LREAL#19.579149162561258, LREAL#19.593929605703352, LREAL#19.608190954002232, LREAL#19.62195143826828, LREAL#19.635228649038805, LREAL#19.648039559064692, LREAL#19.660400545007292, LREAL#19.672327408373313, LREAL#19.683835395714475, LREAL#19.694939218117742, LREAL#19.705653070011053, LREAL#19.715990647308583, LREAL#19.725965164918737, LREAL#19.735589373637257, LREAL#19.74487557644704, LREAL#19.753835644245491, LREAL#19.762481031019547, LREAL#19.77082278848771, LREAL#19.778871580227889, LREAL#19.786637695309036, LREAL#19.794131061444048, LREAL#18.854802175821771, LREAL#18.895021963501684, LREAL#18.933829216781984, LREAL#18.971273544413613, LREAL#19.00740281286912, LREAL#19.042263207532141, LREAL#19.075899291737894, LREAL#19.108354063740133, LREAL#19.13966901167742, LREAL#19.169884166608945, LREAL#19.199038153687717, LREAL#19.227168241536525, LREAL#19.25431038988981, LREAL#19.280499295562311, LREAL#19.305768436803309, LREAL#19.330150116093094, LREAL#19.353675501436445, LREAL#19.37637466620583, LREAL#19.398276627585318, LREAL#19.419409383664327, LREAL#19.439799949228611, LREAL#19.459474390294268, LREAL#19.478457857428893, LREAL#19.496774617902481, LREAL#19.514448086709184, LREAL#19.531500856499555, LREAL#19.54795472646158, LREAL#19.563830730187384, LREAL#19.579149162561258, LREAL#19.593929605703352, LREAL#19.608190954002232, LREAL#19.62195143826828, LREAL#19.635228649038805, LREAL#19.648039559064692, LREAL#19.660400545007292, LREAL#19.672327408373313, LREAL#19.683835395714475, LREAL#19.694939218117742, LREAL#19.705653070011053, LREAL#19.715990647308583, LREAL#19.725965164918737, LREAL#19.735589373637257, LREAL#19.74487557644704, LREAL#19.753835644245491, LREAL#19.762481031019547, LREAL#19.77082278848771, LREAL#19.778871580227889, LREAL#19.786637695309036, LREAL#19.794131061444048, LREAL#19.801361257680728, LREAL#18.895021963501684, LREAL#18.933829216781984, LREAL#18.971273544413613, LREAL#19.00740281286912, LREAL#19.042263207532141, LREAL#19.075899291737894, LREAL#19.108354063740133, LREAL#19.13966901167742, LREAL#19.169884166608945, LREAL#19.199038153687717, LREAL#19.227168241536525, LREAL#19.25431038988981, LREAL#19.280499295562311, LREAL#19.305768436803309, LREAL#19.330150116093094, LREAL#19.353675501436445, LREAL#19.37637466620583, LREAL#19.398276627585318, LREAL#19.419409383664327, LREAL#19.439799949228611, LREAL#19.459474390294268, LREAL#19.478457857428893, LREAL#19.496774617902481, LREAL#19.514448086709184, LREAL#19.531500856499555, LREAL#19.54795472646158, LREAL#19.563830730187384, LREAL#19.579149162561258, LREAL#19.593929605703352, LREAL#19.608190954002232, LREAL#19.62195143826828, LREAL#19.635228649038805, LREAL#19.648039559064692, LREAL#19.660400545007292, LREAL#19.672327408373313, LREAL#19.683835395714475, LREAL#19.694939218117742, LREAL#19.705653070011053, LREAL#19.715990647308583, LREAL#19.725965164918737, LREAL#19.735589373637257, LREAL#19.74487557644704, LREAL#19.753835644245491, LREAL#19.762481031019547, LREAL#19.77082278848771, LREAL#19.778871580227889, LREAL#19.786637695309036, LREAL#19.794131061444048, LREAL#19.801361257680728, LREAL#19.808337526647041, LREAL#18.933829216781984, LREAL#18.971273544413613, LREAL#19.00740281286912, LREAL#19.042263207532141, LREAL#19.075899291737894, LREAL#19.108354063740133, LREAL#19.13966901167742, LREAL#19.169884166608945, LREAL#19.199038153687717, LREAL#19.227168241536525, LREAL#19.25431038988981, LREAL#19.280499295562311, LREAL#19.305768436803309, LREAL#19.330150116093094, LREAL#19.353675501436445, LREAL#19.37637466620583, LREAL#19.398276627585318, LREAL#19.419409383664327, LREAL#19.439799949228611, LREAL#19.459474390294268, LREAL#19.478457857428893, LREAL#19.496774617902481, LREAL#19.514448086709184, LREAL#19.531500856499555, LREAL#19.54795472646158, LREAL#19.563830730187384, LREAL#19.579149162561258, LREAL#19.593929605703352, LREAL#19.608190954002232, LREAL#19.62195143826828, LREAL#19.635228649038805, LREAL#19.648039559064692, LREAL#19.660400545007292, LREAL#19.672327408373313, LREAL#19.683835395714475, LREAL#19.694939218117742, LREAL#19.705653070011053, LREAL#19.715990647308583, LREAL#19.725965164918737, LREAL#19.735589373637257, LREAL#19.74487557644704, LREAL#19.753835644245491, LREAL#19.762481031019547, LREAL#19.77082278848771, LREAL#19.778871580227889, LREAL#19.786637695309036, LREAL#19.794131061444048, LREAL#19.801361257680728, LREAL#19.808337526647041, LREAL#19.815068786366307, LREAL#18.971273544413613, LREAL#19.00740281286912, LREAL#19.042263207532141, LREAL#19.075899291737894, LREAL#19.108354063740133, LREAL#19.13966901167742, LREAL#19.169884166608945, LREAL#19.199038153687717, LREAL#19.227168241536525, LREAL#19.25431038988981, LREAL#19.280499295562311, LREAL#19.305768436803309, LREAL#19.330150116093094, LREAL#19.353675501436445, LREAL#19.37637466620583, LREAL#19.398276627585318, LREAL#19.419409383664327, LREAL#19.439799949228611, LREAL#19.459474390294268, LREAL#19.478457857428893, LREAL#19.496774617902481, LREAL#19.514448086709184, LREAL#19.531500856499555, LREAL#19.54795472646158, LREAL#19.563830730187384, LREAL#19.579149162561258, LREAL#19.593929605703352, LREAL#19.608190954002232, LREAL#19.62195143826828, LREAL#19.635228649038805, LREAL#19.648039559064692, LREAL#19.660400545007292, LREAL#19.672327408373313, LREAL#19.683835395714475, LREAL#19.694939218117742, LREAL#19.705653070011053, LREAL#19.715990647308583, LREAL#19.725965164918737, LREAL#19.735589373637257, LREAL#19.74487557644704, LREAL#19.753835644245491, LREAL#19.762481031019547, LREAL#19.77082278848771, LREAL#19.778871580227889, LREAL#19.786637695309036, LREAL#19.794131061444048, LREAL#19.801361257680728, LREAL#19.808337526647041, LREAL#19.815068786366307, LREAL#19.821563641657438, LREAL#19.00740281286912, LREAL#19.042263207532141, LREAL#19.075899291737894, LREAL#19.108354063740133, LREAL#19.13966901167742, LREAL#19.169884166608945, LREAL#19.199038153687717, LREAL#19.227168241536525, LREAL#19.25431038988981, LREAL#19.280499295562311, LREAL#19.305768436803309, LREAL#19.330150116093094, LREAL#19.353675501436445, LREAL#19.37637466620583, LREAL#19.398276627585318, LREAL#19.419409383664327, LREAL#19.439799949228611, LREAL#19.459474390294268, LREAL#19.478457857428893, LREAL#19.496774617902481, LREAL#19.514448086709184, LREAL#19.531500856499555, LREAL#19.54795472646158, LREAL#19.563830730187384, LREAL#19.579149162561258, LREAL#19.593929605703352, LREAL#19.608190954002232, LREAL#19.62195143826828, LREAL#19.635228649038805, LREAL#19.648039559064692, LREAL#19.660400545007292, LREAL#19.672327408373313, LREAL#19.683835395714475, LREAL#19.694939218117742, LREAL#19.705653070011053, LREAL#19.715990647308583, LREAL#19.725965164918737, LREAL#19.735589373637257, LREAL#19.74487557644704, LREAL#19.753835644245491, LREAL#19.762481031019547, LREAL#19.77082278848771, LREAL#19.778871580227889, LREAL#19.786637695309036, LREAL#19.794131061444048, LREAL#19.801361257680728, LREAL#19.808337526647041, LREAL#19.815068786366307, LREAL#19.821563641657438, LREAL#19.827830395134797, LREAL#19.042263207532141, LREAL#19.075899291737894, LREAL#19.108354063740133, LREAL#19.13966901167742, LREAL#19.169884166608945, LREAL#19.199038153687717, LREAL#19.227168241536525, LREAL#19.25431038988981, LREAL#19.280499295562311, LREAL#19.305768436803309, LREAL#19.330150116093094, LREAL#19.353675501436445, LREAL#19.37637466620583, LREAL#19.398276627585318, LREAL#19.419409383664327, LREAL#19.439799949228611, LREAL#19.459474390294268, LREAL#19.478457857428893, LREAL#19.496774617902481, LREAL#19.514448086709184, LREAL#19.531500856499555, LREAL#19.54795472646158, LREAL#19.563830730187384, LREAL#19.579149162561258, LREAL#19.593929605703352, LREAL#19.608190954002232, LREAL#19.62195143826828, LREAL#19.635228649038805, LREAL#19.648039559064692, LREAL#19.660400545007292, LREAL#19.672327408373313, LREAL#19.683835395714475, LREAL#19.694939218117742, LREAL#19.705653070011053, LREAL#19.715990647308583, LREAL#19.725965164918737, LREAL#19.735589373637257, LREAL#19.74487557644704, LREAL#19.753835644245491, LREAL#19.762481031019547, LREAL#19.77082278848771, LREAL#19.778871580227889, LREAL#19.786637695309036, LREAL#19.794131061444048, LREAL#19.801361257680728, LREAL#19.808337526647041, LREAL#19.815068786366307, LREAL#19.821563641657438, LREAL#19.827830395134797, LREAL#19.833877057821745, LREAL#19.075899291737894, LREAL#19.108354063740133, LREAL#19.13966901167742, LREAL#19.169884166608945, LREAL#19.199038153687717, LREAL#19.227168241536525, LREAL#19.25431038988981, LREAL#19.280499295562311, LREAL#19.305768436803309, LREAL#19.330150116093094, LREAL#19.353675501436445, LREAL#19.37637466620583, LREAL#19.398276627585318, LREAL#19.419409383664327, LREAL#19.439799949228611, LREAL#19.459474390294268, LREAL#19.478457857428893, LREAL#19.496774617902481, LREAL#19.514448086709184, LREAL#19.531500856499555, LREAL#19.54795472646158, LREAL#19.563830730187384, LREAL#19.579149162561258, LREAL#19.593929605703352, LREAL#19.608190954002232, LREAL#19.62195143826828, LREAL#19.635228649038805, LREAL#19.648039559064692, LREAL#19.660400545007292, LREAL#19.672327408373313, LREAL#19.683835395714475, LREAL#19.694939218117742, LREAL#19.705653070011053, LREAL#19.715990647308583, LREAL#19.725965164918737, LREAL#19.735589373637257, LREAL#19.74487557644704, LREAL#19.753835644245491, LREAL#19.762481031019547, LREAL#19.77082278848771, LREAL#19.778871580227889, LREAL#19.786637695309036, LREAL#19.794131061444048, LREAL#19.801361257680728, LREAL#19.808337526647041, LREAL#19.815068786366307, LREAL#19.821563641657438, LREAL#19.827830395134797, LREAL#19.833877057821745, LREAL#19.839711359391419, LREAL#19.108354063740133, LREAL#19.13966901167742, LREAL#19.169884166608945, LREAL#19.199038153687717, LREAL#19.227168241536525, LREAL#19.25431038988981, LREAL#19.280499295562311, LREAL#19.305768436803309, LREAL#19.330150116093094, LREAL#19.353675501436445, LREAL#19.37637466620583, LREAL#19.398276627585318, LREAL#19.419409383664327, LREAL#19.439799949228611, LREAL#19.459474390294268, LREAL#19.478457857428893, LREAL#19.496774617902481, LREAL#19.514448086709184, LREAL#19.531500856499555, LREAL#19.54795472646158, LREAL#19.563830730187384, LREAL#19.579149162561258, LREAL#19.593929605703352, LREAL#19.608190954002232, LREAL#19.62195143826828, LREAL#19.635228649038805, LREAL#19.648039559064692, LREAL#19.660400545007292, LREAL#19.672327408373313, LREAL#19.683835395714475, LREAL#19.694939218117742, LREAL#19.705653070011053, LREAL#19.715990647308583, LREAL#19.725965164918737, LREAL#19.735589373637257, LREAL#19.74487557644704, LREAL#19.753835644245491, LREAL#19.762481031019547, LREAL#19.77082278848771, LREAL#19.778871580227889, LREAL#19.786637695309036, LREAL#19.794131061444048, LREAL#19.801361257680728, LREAL#19.808337526647041, LREAL#19.815068786366307, LREAL#19.821563641657438, LREAL#19.827830395134797, LREAL#19.833877057821745, LREAL#19.839711359391419, LREAL#19.845340758047868, LREAL#19.13966901167742, LREAL#19.169884166608945, LREAL#19.199038153687717, LREAL#19.227168241536525, LREAL#19.25431038988981, LREAL#19.280499295562311, LREAL#19.305768436803309, LREAL#19.330150116093094, LREAL#19.353675501436445, LREAL#19.37637466620583, LREAL#19.398276627585318, LREAL#19.419409383664327, LREAL#19.439799949228611, LREAL#19.459474390294268, LREAL#19.478457857428893, LREAL#19.496774617902481, LREAL#19.514448086709184, LREAL#19.531500856499555, LREAL#19.54795472646158, LREAL#19.563830730187384, LREAL#19.579149162561258, LREAL#19.593929605703352, LREAL#19.608190954002232, LREAL#19.62195143826828, LREAL#19.635228649038805, LREAL#19.648039559064692, LREAL#19.660400545007292, LREAL#19.672327408373313, LREAL#19.683835395714475, LREAL#19.694939218117742, LREAL#19.705653070011053, LREAL#19.715990647308583, LREAL#19.725965164918737, LREAL#19.735589373637257, LREAL#19.74487557644704, LREAL#19.753835644245491, LREAL#19.762481031019547, LREAL#19.77082278848771, LREAL#19.778871580227889, LREAL#19.786637695309036, LREAL#19.794131061444048, LREAL#19.801361257680728, LREAL#19.808337526647041, LREAL#19.815068786366307, LREAL#19.821563641657438, LREAL#19.827830395134797, LREAL#19.833877057821745, LREAL#19.839711359391419, LREAL#19.845340758047868, LREAL#19.850772450060148, LREAL#19.169884166608945, LREAL#19.199038153687717, LREAL#19.227168241536525, LREAL#19.25431038988981, LREAL#19.280499295562311, LREAL#19.305768436803309, LREAL#19.330150116093094, LREAL#19.353675501436445, LREAL#19.37637466620583, LREAL#19.398276627585318, LREAL#19.419409383664327, LREAL#19.439799949228611, LREAL#19.459474390294268, LREAL#19.478457857428893, LREAL#19.496774617902481, LREAL#19.514448086709184, LREAL#19.531500856499555, LREAL#19.54795472646158, LREAL#19.563830730187384, LREAL#19.579149162561258, LREAL#19.593929605703352, LREAL#19.608190954002232, LREAL#19.62195143826828, LREAL#19.635228649038805, LREAL#19.648039559064692, LREAL#19.660400545007292, LREAL#19.672327408373313, LREAL#19.683835395714475, LREAL#19.694939218117742, LREAL#19.705653070011053, LREAL#19.715990647308583, LREAL#19.725965164918737, LREAL#19.735589373637257, LREAL#19.74487557644704, LREAL#19.753835644245491, LREAL#19.762481031019547, LREAL#19.77082278848771, LREAL#19.778871580227889, LREAL#19.786637695309036, LREAL#19.794131061444048, LREAL#19.801361257680728, LREAL#19.808337526647041, LREAL#19.815068786366307, LREAL#19.821563641657438, LREAL#19.827830395134797, LREAL#19.833877057821745, LREAL#19.839711359391419, LREAL#19.845340758047868, LREAL#19.850772450060148, LREAL#19.856013378961581, LREAL#19.199038153687717, LREAL#19.227168241536525, LREAL#19.25431038988981, LREAL#19.280499295562311, LREAL#19.305768436803309, LREAL#19.330150116093094, LREAL#19.353675501436445, LREAL#19.37637466620583, LREAL#19.398276627585318, LREAL#19.419409383664327, LREAL#19.439799949228611, LREAL#19.459474390294268, LREAL#19.478457857428893, LREAL#19.496774617902481, LREAL#19.514448086709184, LREAL#19.531500856499555, LREAL#19.54795472646158, LREAL#19.563830730187384, LREAL#19.579149162561258, LREAL#19.593929605703352, LREAL#19.608190954002232, LREAL#19.62195143826828, LREAL#19.635228649038805, LREAL#19.648039559064692, LREAL#19.660400545007292, LREAL#19.672327408373313, LREAL#19.683835395714475, LREAL#19.694939218117742, LREAL#19.705653070011053, LREAL#19.715990647308583, LREAL#19.725965164918737, LREAL#19.735589373637257, LREAL#19.74487557644704, LREAL#19.753835644245491, LREAL#19.762481031019547, LREAL#19.77082278848771, LREAL#19.778871580227889, LREAL#19.786637695309036, LREAL#19.794131061444048, LREAL#19.801361257680728, LREAL#19.808337526647041, LREAL#19.815068786366307, LREAL#19.821563641657438, LREAL#19.827830395134797, LREAL#19.833877057821745, LREAL#19.839711359391419, LREAL#19.845340758047868, LREAL#19.850772450060148, LREAL#19.856013378961581, LREAL#19.861070244425928, LREAL#19.227168241536525, LREAL#19.25431038988981, LREAL#19.280499295562311, LREAL#19.305768436803309, LREAL#19.330150116093094, LREAL#19.353675501436445, LREAL#19.37637466620583, LREAL#19.398276627585318, LREAL#19.419409383664327, LREAL#19.439799949228611, LREAL#19.459474390294268, LREAL#19.478457857428893, LREAL#19.496774617902481, LREAL#19.514448086709184, LREAL#19.531500856499555, LREAL#19.54795472646158, LREAL#19.563830730187384, LREAL#19.579149162561258, LREAL#19.593929605703352, LREAL#19.608190954002232, LREAL#19.62195143826828, LREAL#19.635228649038805, LREAL#19.648039559064692, LREAL#19.660400545007292, LREAL#19.672327408373313, LREAL#19.683835395714475, LREAL#19.694939218117742, LREAL#19.705653070011053, LREAL#19.715990647308583, LREAL#19.725965164918737, LREAL#19.735589373637257, LREAL#19.74487557644704, LREAL#19.753835644245491, LREAL#19.762481031019547, LREAL#19.77082278848771, LREAL#19.778871580227889, LREAL#19.786637695309036, LREAL#19.794131061444048, LREAL#19.801361257680728, LREAL#19.808337526647041, LREAL#19.815068786366307, LREAL#19.821563641657438, LREAL#19.827830395134797, LREAL#19.833877057821745, LREAL#19.839711359391419, LREAL#19.845340758047868, LREAL#19.850772450060148, LREAL#19.856013378961581, LREAL#19.861070244425928, LREAL#19.865949510831836, LREAL#19.25431038988981, LREAL#19.280499295562311, LREAL#19.305768436803309, LREAL#19.330150116093094, LREAL#19.353675501436445, LREAL#19.37637466620583, LREAL#19.398276627585318, LREAL#19.419409383664327, LREAL#19.439799949228611, LREAL#19.459474390294268, LREAL#19.478457857428893, LREAL#19.496774617902481, LREAL#19.514448086709184, LREAL#19.531500856499555, LREAL#19.54795472646158, LREAL#19.563830730187384, LREAL#19.579149162561258, LREAL#19.593929605703352, LREAL#19.608190954002232, LREAL#19.62195143826828, LREAL#19.635228649038805, LREAL#19.648039559064692, LREAL#19.660400545007292, LREAL#19.672327408373313, LREAL#19.683835395714475, LREAL#19.694939218117742, LREAL#19.705653070011053, LREAL#19.715990647308583, LREAL#19.725965164918737, LREAL#19.735589373637257, LREAL#19.74487557644704, LREAL#19.753835644245491, LREAL#19.762481031019547, LREAL#19.77082278848771, LREAL#19.778871580227889, LREAL#19.786637695309036, LREAL#19.794131061444048, LREAL#19.801361257680728, LREAL#19.808337526647041, LREAL#19.815068786366307, LREAL#19.821563641657438, LREAL#19.827830395134797, LREAL#19.833877057821745, LREAL#19.839711359391419, LREAL#19.845340758047868, LREAL#19.850772450060148, LREAL#19.856013378961581, LREAL#19.861070244425928, LREAL#19.865949510831836, LREAL#19.870657415526487, LREAL#19.280499295562311, LREAL#19.305768436803309, LREAL#19.330150116093094, LREAL#19.353675501436445, LREAL#19.37637466620583, LREAL#19.398276627585318, LREAL#19.419409383664327, LREAL#19.439799949228611, LREAL#19.459474390294268, LREAL#19.478457857428893, LREAL#19.496774617902481, LREAL#19.514448086709184, LREAL#19.531500856499555, LREAL#19.54795472646158, LREAL#19.563830730187384, LREAL#19.579149162561258, LREAL#19.593929605703352, LREAL#19.608190954002232, LREAL#19.62195143826828, LREAL#19.635228649038805, LREAL#19.648039559064692, LREAL#19.660400545007292, LREAL#19.672327408373313, LREAL#19.683835395714475, LREAL#19.694939218117742, LREAL#19.705653070011053, LREAL#19.715990647308583, LREAL#19.725965164918737, LREAL#19.735589373637257, LREAL#19.74487557644704, LREAL#19.753835644245491, LREAL#19.762481031019547, LREAL#19.77082278848771, LREAL#19.778871580227889, LREAL#19.786637695309036, LREAL#19.794131061444048, LREAL#19.801361257680728, LREAL#19.808337526647041, LREAL#19.815068786366307, LREAL#19.821563641657438, LREAL#19.827830395134797, LREAL#19.833877057821745, LREAL#19.839711359391419, LREAL#19.845340758047868, LREAL#19.850772450060148, LREAL#19.856013378961581, LREAL#19.861070244425928, LREAL#19.865949510831836, LREAL#19.870657415526487, LREAL#19.875199976799031, LREAL#19.305768436803309, LREAL#19.330150116093094, LREAL#19.353675501436445, LREAL#19.37637466620583, LREAL#19.398276627585318, LREAL#19.419409383664327, LREAL#19.439799949228611, LREAL#19.459474390294268, LREAL#19.478457857428893, LREAL#19.496774617902481, LREAL#19.514448086709184, LREAL#19.531500856499555, LREAL#19.54795472646158, LREAL#19.563830730187384, LREAL#19.579149162561258, LREAL#19.593929605703352, LREAL#19.608190954002232, LREAL#19.62195143826828, LREAL#19.635228649038805, LREAL#19.648039559064692, LREAL#19.660400545007292, LREAL#19.672327408373313, LREAL#19.683835395714475, LREAL#19.694939218117742, LREAL#19.705653070011053, LREAL#19.715990647308583, LREAL#19.725965164918737, LREAL#19.735589373637257, LREAL#19.74487557644704, LREAL#19.753835644245491, LREAL#19.762481031019547, LREAL#19.77082278848771, LREAL#19.778871580227889, LREAL#19.786637695309036, LREAL#19.794131061444048, LREAL#19.801361257680728, LREAL#19.808337526647041, LREAL#19.815068786366307, LREAL#19.821563641657438, LREAL#19.827830395134797, LREAL#19.833877057821745, LREAL#19.839711359391419, LREAL#19.845340758047868, LREAL#19.850772450060148, LREAL#19.856013378961581, LREAL#19.861070244425928, LREAL#19.865949510831836, LREAL#19.870657415526487, LREAL#19.875199976799031, LREAL#19.879583001573998, LREAL#19.330150116093094, LREAL#19.353675501436445, LREAL#19.37637466620583, LREAL#19.398276627585318, LREAL#19.419409383664327, LREAL#19.439799949228611, LREAL#19.459474390294268, LREAL#19.478457857428893, LREAL#19.496774617902481, LREAL#19.514448086709184, LREAL#19.531500856499555, LREAL#19.54795472646158, LREAL#19.563830730187384, LREAL#19.579149162561258, LREAL#19.593929605703352, LREAL#19.608190954002232, LREAL#19.62195143826828, LREAL#19.635228649038805, LREAL#19.648039559064692, LREAL#19.660400545007292, LREAL#19.672327408373313, LREAL#19.683835395714475, LREAL#19.694939218117742, LREAL#19.705653070011053, LREAL#19.715990647308583, LREAL#19.725965164918737, LREAL#19.735589373637257, LREAL#19.74487557644704, LREAL#19.753835644245491, LREAL#19.762481031019547, LREAL#19.77082278848771, LREAL#19.778871580227889, LREAL#19.786637695309036, LREAL#19.794131061444048, LREAL#19.801361257680728, LREAL#19.808337526647041, LREAL#19.815068786366307, LREAL#19.821563641657438, LREAL#19.827830395134797, LREAL#19.833877057821745, LREAL#19.839711359391419, LREAL#19.845340758047868, LREAL#19.850772450060148, LREAL#19.856013378961581, LREAL#19.861070244425928, LREAL#19.865949510831836, LREAL#19.870657415526487, LREAL#19.875199976799031, LREAL#19.879583001573998, LREAL#19.883812092834489, LREAL#19.353675501436445, LREAL#19.37637466620583, LREAL#19.398276627585318, LREAL#19.419409383664327, LREAL#19.439799949228611, LREAL#19.459474390294268, LREAL#19.478457857428893, LREAL#19.496774617902481, LREAL#19.514448086709184, LREAL#19.531500856499555, LREAL#19.54795472646158, LREAL#19.563830730187384, LREAL#19.579149162561258, LREAL#19.593929605703352, LREAL#19.608190954002232, LREAL#19.62195143826828, LREAL#19.635228649038805, LREAL#19.648039559064692, LREAL#19.660400545007292, LREAL#19.672327408373313, LREAL#19.683835395714475, LREAL#19.694939218117742, LREAL#19.705653070011053, LREAL#19.715990647308583, LREAL#19.725965164918737, LREAL#19.735589373637257, LREAL#19.74487557644704, LREAL#19.753835644245491, LREAL#19.762481031019547, LREAL#19.77082278848771, LREAL#19.778871580227889, LREAL#19.786637695309036, LREAL#19.794131061444048, LREAL#19.801361257680728, LREAL#19.808337526647041, LREAL#19.815068786366307, LREAL#19.821563641657438, LREAL#19.827830395134797, LREAL#19.833877057821745, LREAL#19.839711359391419, LREAL#19.845340758047868, LREAL#19.850772450060148, LREAL#19.856013378961581, LREAL#19.861070244425928, LREAL#19.865949510831836, LREAL#19.870657415526487, LREAL#19.875199976799031, LREAL#19.879583001573998, LREAL#19.883812092834489, LREAL#19.88789265678469, LREAL#19.37637466620583, LREAL#19.398276627585318, LREAL#19.419409383664327, LREAL#19.439799949228611, LREAL#19.459474390294268, LREAL#19.478457857428893, LREAL#19.496774617902481, LREAL#19.514448086709184, LREAL#19.531500856499555, LREAL#19.54795472646158, LREAL#19.563830730187384, LREAL#19.579149162561258, LREAL#19.593929605703352, LREAL#19.608190954002232, LREAL#19.62195143826828, LREAL#19.635228649038805, LREAL#19.648039559064692, LREAL#19.660400545007292, LREAL#19.672327408373313, LREAL#19.683835395714475, LREAL#19.694939218117742, LREAL#19.705653070011053, LREAL#19.715990647308583, LREAL#19.725965164918737, LREAL#19.735589373637257, LREAL#19.74487557644704, LREAL#19.753835644245491, LREAL#19.762481031019547, LREAL#19.77082278848771, LREAL#19.778871580227889, LREAL#19.786637695309036, LREAL#19.794131061444048, LREAL#19.801361257680728, LREAL#19.808337526647041, LREAL#19.815068786366307, LREAL#19.821563641657438, LREAL#19.827830395134797, LREAL#19.833877057821745, LREAL#19.839711359391419, LREAL#19.845340758047868, LREAL#19.850772450060148, LREAL#19.856013378961581, LREAL#19.861070244425928, LREAL#19.865949510831836, LREAL#19.870657415526487, LREAL#19.875199976799031, LREAL#19.879583001573998, LREAL#19.883812092834489, LREAL#19.88789265678469, LREAL#19.891829909760816, LREAL#19.398276627585318, LREAL#19.419409383664327, LREAL#19.439799949228611, LREAL#19.459474390294268, LREAL#19.478457857428893, LREAL#19.496774617902481, LREAL#19.514448086709184, LREAL#19.531500856499555, LREAL#19.54795472646158, LREAL#19.563830730187384, LREAL#19.579149162561258, LREAL#19.593929605703352, LREAL#19.608190954002232, LREAL#19.62195143826828, LREAL#19.635228649038805, LREAL#19.648039559064692, LREAL#19.660400545007292, LREAL#19.672327408373313, LREAL#19.683835395714475, LREAL#19.694939218117742, LREAL#19.705653070011053, LREAL#19.715990647308583, LREAL#19.725965164918737, LREAL#19.735589373637257, LREAL#19.74487557644704, LREAL#19.753835644245491, LREAL#19.762481031019547, LREAL#19.77082278848771, LREAL#19.778871580227889, LREAL#19.786637695309036, LREAL#19.794131061444048, LREAL#19.801361257680728, LREAL#19.808337526647041, LREAL#19.815068786366307, LREAL#19.821563641657438, LREAL#19.827830395134797, LREAL#19.833877057821745, LREAL#19.839711359391419, LREAL#19.845340758047868, LREAL#19.850772450060148, LREAL#19.856013378961581, LREAL#19.861070244425928, LREAL#19.865949510831836, LREAL#19.870657415526487, LREAL#19.875199976799031, LREAL#19.879583001573998, LREAL#19.883812092834489, LREAL#19.88789265678469, LREAL#19.891829909760816, LREAL#19.895628884899349, LREAL#19.419409383664327, LREAL#19.439799949228611, LREAL#19.459474390294268, LREAL#19.478457857428893, LREAL#19.496774617902481, LREAL#19.514448086709184, LREAL#19.531500856499555, LREAL#19.54795472646158, LREAL#19.563830730187384, LREAL#19.579149162561258, LREAL#19.593929605703352, LREAL#19.608190954002232, LREAL#19.62195143826828, LREAL#19.635228649038805, LREAL#19.648039559064692, LREAL#19.660400545007292, LREAL#19.672327408373313, LREAL#19.683835395714475, LREAL#19.694939218117742, LREAL#19.705653070011053, LREAL#19.715990647308583, LREAL#19.725965164918737, LREAL#19.735589373637257, LREAL#19.74487557644704, LREAL#19.753835644245491, LREAL#19.762481031019547, LREAL#19.77082278848771, LREAL#19.778871580227889, LREAL#19.786637695309036, LREAL#19.794131061444048, LREAL#19.801361257680728, LREAL#19.808337526647041, LREAL#19.815068786366307, LREAL#19.821563641657438, LREAL#19.827830395134797, LREAL#19.833877057821745, LREAL#19.839711359391419, LREAL#19.845340758047868, LREAL#19.850772450060148, LREAL#19.856013378961581, LREAL#19.861070244425928, LREAL#19.865949510831836, LREAL#19.870657415526487, LREAL#19.875199976799031, LREAL#19.879583001573998, LREAL#19.883812092834489, LREAL#19.88789265678469, LREAL#19.891829909760816, LREAL#19.895628884899349, LREAL#19.899294438571086, LREAL#19.439799949228611, LREAL#19.459474390294268, LREAL#19.478457857428893, LREAL#19.496774617902481, LREAL#19.514448086709184, LREAL#19.531500856499555, LREAL#19.54795472646158, LREAL#19.563830730187384, LREAL#19.579149162561258, LREAL#19.593929605703352, LREAL#19.608190954002232, LREAL#19.62195143826828, LREAL#19.635228649038805, LREAL#19.648039559064692, LREAL#19.660400545007292, LREAL#19.672327408373313, LREAL#19.683835395714475, LREAL#19.694939218117742, LREAL#19.705653070011053, LREAL#19.715990647308583, LREAL#19.725965164918737, LREAL#19.735589373637257, LREAL#19.74487557644704, LREAL#19.753835644245491, LREAL#19.762481031019547, LREAL#19.77082278848771, LREAL#19.778871580227889, LREAL#19.786637695309036, LREAL#19.794131061444048, LREAL#19.801361257680728, LREAL#19.808337526647041, LREAL#19.815068786366307, LREAL#19.821563641657438, LREAL#19.827830395134797, LREAL#19.833877057821745, LREAL#19.839711359391419, LREAL#19.845340758047868, LREAL#19.850772450060148, LREAL#19.856013378961581, LREAL#19.861070244425928, LREAL#19.865949510831836, LREAL#19.870657415526487, LREAL#19.875199976799031, LREAL#19.879583001573998, LREAL#19.883812092834489, LREAL#19.88789265678469, LREAL#19.891829909760816, LREAL#19.895628884899349, LREAL#19.899294438571086, LREAL#19.902831256589216, LREAL#19.459474390294268, LREAL#19.478457857428893, LREAL#19.496774617902481, LREAL#19.514448086709184, LREAL#19.531500856499555, LREAL#19.54795472646158, LREAL#19.563830730187384, LREAL#19.579149162561258, LREAL#19.593929605703352, LREAL#19.608190954002232, LREAL#19.62195143826828, LREAL#19.635228649038805, LREAL#19.648039559064692, LREAL#19.660400545007292, LREAL#19.672327408373313, LREAL#19.683835395714475, LREAL#19.694939218117742, LREAL#19.705653070011053, LREAL#19.715990647308583, LREAL#19.725965164918737, LREAL#19.735589373637257, LREAL#19.74487557644704, LREAL#19.753835644245491, LREAL#19.762481031019547, LREAL#19.77082278848771, LREAL#19.778871580227889, LREAL#19.786637695309036, LREAL#19.794131061444048, LREAL#19.801361257680728, LREAL#19.808337526647041, LREAL#19.815068786366307, LREAL#19.821563641657438, LREAL#19.827830395134797, LREAL#19.833877057821745, LREAL#19.839711359391419, LREAL#19.845340758047868, LREAL#19.850772450060148, LREAL#19.856013378961581, LREAL#19.861070244425928, LREAL#19.865949510831836, LREAL#19.870657415526487, LREAL#19.875199976799031, LREAL#19.879583001573998, LREAL#19.883812092834489, LREAL#19.88789265678469, LREAL#19.891829909760816, LREAL#19.895628884899349, LREAL#19.899294438571086, LREAL#19.902831256589216, LREAL#0.0, LREAL#19.478457857428893, LREAL#19.496774617902481, LREAL#19.514448086709184, LREAL#19.531500856499555, LREAL#19.54795472646158, LREAL#19.563830730187384, LREAL#19.579149162561258, LREAL#19.593929605703352, LREAL#19.608190954002232, LREAL#19.62195143826828, LREAL#19.635228649038805, LREAL#19.648039559064692, LREAL#19.660400545007292, LREAL#19.672327408373313, LREAL#19.683835395714475, LREAL#19.694939218117742, LREAL#19.705653070011053, LREAL#19.715990647308583, LREAL#19.725965164918737, LREAL#19.735589373637257, LREAL#19.74487557644704, LREAL#19.753835644245491, LREAL#19.762481031019547, LREAL#19.77082278848771, LREAL#19.778871580227889, LREAL#19.786637695309036, LREAL#19.794131061444048, LREAL#19.801361257680728, LREAL#19.808337526647041, LREAL#19.815068786366307, LREAL#19.821563641657438, LREAL#19.827830395134797, LREAL#19.833877057821745, LREAL#19.839711359391419, LREAL#19.845340758047868, LREAL#19.850772450060148, LREAL#19.856013378961581, LREAL#19.861070244425928, LREAL#19.865949510831836, LREAL#19.870657415526487, LREAL#19.875199976799031, LREAL#19.879583001573998, LREAL#19.883812092834489, LREAL#19.88789265678469, LREAL#19.891829909760816, LREAL#19.895628884899349, LREAL#19.899294438571086, LREAL#19.902831256589216, LREAL#0.0, LREAL#0.0, LREAL#19.496774617902481, LREAL#19.514448086709184, LREAL#19.531500856499555, LREAL#19.54795472646158, LREAL#19.563830730187384, LREAL#19.579149162561258, LREAL#19.593929605703352, LREAL#19.608190954002232, LREAL#19.62195143826828, LREAL#19.635228649038805, LREAL#19.648039559064692, LREAL#19.660400545007292, LREAL#19.672327408373313, LREAL#19.683835395714475, LREAL#19.694939218117742, LREAL#19.705653070011053, LREAL#19.715990647308583, LREAL#19.725965164918737, LREAL#19.735589373637257, LREAL#19.74487557644704, LREAL#19.753835644245491, LREAL#19.762481031019547, LREAL#19.77082278848771, LREAL#19.778871580227889, LREAL#19.786637695309036, LREAL#19.794131061444048, LREAL#19.801361257680728, LREAL#19.808337526647041, LREAL#19.815068786366307, LREAL#19.821563641657438, LREAL#19.827830395134797, LREAL#19.833877057821745, LREAL#19.839711359391419, LREAL#19.845340758047868, LREAL#19.850772450060148, LREAL#19.856013378961581, LREAL#19.861070244425928, LREAL#19.865949510831836, LREAL#19.870657415526487, LREAL#19.875199976799031, LREAL#19.879583001573998, LREAL#19.883812092834489, LREAL#19.88789265678469, LREAL#19.891829909760816, LREAL#19.895628884899349, LREAL#19.899294438571086, LREAL#19.902831256589216, LREAL#0.0, LREAL#0.0, LREAL#0.0, LREAL#19.514448086709184, LREAL#19.531500856499555, LREAL#19.54795472646158, LREAL#19.563830730187384, LREAL#19.579149162561258, LREAL#19.593929605703352, LREAL#19.608190954002232, LREAL#19.62195143826828, LREAL#19.635228649038805, LREAL#19.648039559064692, LREAL#19.660400545007292, LREAL#19.672327408373313, LREAL#19.683835395714475, LREAL#19.694939218117742, LREAL#19.705653070011053, LREAL#19.715990647308583, LREAL#19.725965164918737, LREAL#19.735589373637257, LREAL#19.74487557644704, LREAL#19.753835644245491, LREAL#19.762481031019547, LREAL#19.77082278848771, LREAL#19.778871580227889, LREAL#19.786637695309036, LREAL#19.794131061444048, LREAL#19.801361257680728, LREAL#19.808337526647041, LREAL#19.815068786366307, LREAL#19.821563641657438, LREAL#19.827830395134797, LREAL#19.833877057821745, LREAL#19.839711359391419, LREAL#19.845340758047868, LREAL#19.850772450060148, LREAL#19.856013378961581, LREAL#19.861070244425928, LREAL#19.865949510831836, LREAL#19.870657415526487, LREAL#19.875199976799031, LREAL#19.879583001573998, LREAL#19.883812092834489, LREAL#19.88789265678469, LREAL#19.891829909760816, LREAL#19.895628884899349, LREAL#19.899294438571086, LREAL#19.902831256589216, LREAL#0.0, LREAL#0.0, LREAL#0.0, LREAL#0.0, LREAL#19.531500856499555, LREAL#19.54795472646158, LREAL#19.563830730187384, LREAL#19.579149162561258, LREAL#19.593929605703352, LREAL#19.608190954002232, LREAL#19.62195143826828, LREAL#19.635228649038805, LREAL#19.648039559064692, LREAL#19.660400545007292, LREAL#19.672327408373313, LREAL#19.683835395714475, LREAL#19.694939218117742, LREAL#19.705653070011053, LREAL#19.715990647308583, LREAL#19.725965164918737, LREAL#19.735589373637257, LREAL#19.74487557644704, LREAL#19.753835644245491, LREAL#19.762481031019547, LREAL#19.77082278848771, LREAL#19.778871580227889, LREAL#19.786637695309036, LREAL#19.794131061444048, LREAL#19.801361257680728, LREAL#19.808337526647041, LREAL#19.815068786366307, LREAL#19.821563641657438, LREAL#19.827830395134797, LREAL#19.833877057821745, LREAL#19.839711359391419, LREAL#19.845340758047868, LREAL#19.850772450060148, LREAL#19.856013378961581, LREAL#19.861070244425928, LREAL#19.865949510831836, LREAL#19.870657415526487, LREAL#19.875199976799031, LREAL#19.879583001573998, LREAL#19.883812092834489, LREAL#19.88789265678469, LREAL#19.891829909760816, LREAL#19.895628884899349, LREAL#19.899294438571086, LREAL#19.902831256589216, LREAL#0.0, LREAL#0.0, LREAL#0.0, LREAL#0.0, LREAL#0.0, LREAL#19.54795472646158, LREAL#19.563830730187384, LREAL#19.579149162561258, LREAL#19.593929605703352, LREAL#19.608190954002232, LREAL#19.62195143826828, LREAL#19.635228649038805, LREAL#19.648039559064692, LREAL#19.660400545007292, LREAL#19.672327408373313, LREAL#19.683835395714475, LREAL#19.694939218117742, LREAL#19.705653070011053, LREAL#19.715990647308583, LREAL#19.725965164918737, LREAL#19.735589373637257, LREAL#19.74487557644704, LREAL#19.753835644245491, LREAL#19.762481031019547, LREAL#19.77082278848771, LREAL#19.778871580227889, LREAL#19.786637695309036, LREAL#19.794131061444048, LREAL#19.801361257680728, LREAL#19.808337526647041, LREAL#19.815068786366307, LREAL#19.821563641657438, LREAL#19.827830395134797, LREAL#19.833877057821745, LREAL#19.839711359391419, LREAL#19.845340758047868, LREAL#19.850772450060148, LREAL#19.856013378961581, LREAL#19.861070244425928, LREAL#19.865949510831836, LREAL#19.870657415526487, LREAL#19.875199976799031, LREAL#19.879583001573998, LREAL#19.883812092834489, LREAL#19.88789265678469, LREAL#19.891829909760816, LREAL#19.895628884899349, LREAL#19.899294438571086, LREAL#19.902831256589216, LREAL#0.0, LREAL#0.0, LREAL#0.0, LREAL#0.0, LREAL#0.0, LREAL#0.0, LREAL#19.563830730187384, LREAL#19.579149162561258, LREAL#19.593929605703352, LREAL#19.608190954002232, LREAL#19.62195143826828, LREAL#19.635228649038805, LREAL#19.648039559064692, LREAL#19.660400545007292, LREAL#19.672327408373313, LREAL#19.683835395714475, LREAL#19.694939218117742, LREAL#19.705653070011053, LREAL#19.715990647308583, LREAL#19.725965164918737, LREAL#19.735589373637257, LREAL#19.74487557644704, LREAL#19.753835644245491, LREAL#19.762481031019547, LREAL#19.77082278848771, LREAL#19.778871580227889, LREAL#19.786637695309036, LREAL#19.794131061444048, LREAL#19.801361257680728, LREAL#19.808337526647041, LREAL#19.815068786366307, LREAL#19.821563641657438, LREAL#19.827830395134797, LREAL#19.833877057821745, LREAL#19.839711359391419, LREAL#19.845340758047868, LREAL#19.850772450060148, LREAL#19.856013378961581, LREAL#19.861070244425928, LREAL#19.865949510831836, LREAL#19.870657415526487, LREAL#19.875199976799031, LREAL#19.879583001573998, LREAL#19.883812092834489, LREAL#19.88789265678469, LREAL#19.891829909760816, LREAL#19.895628884899349, LREAL#19.899294438571086, LREAL#19.902831256589216, LREAL#0.0, LREAL#0.0, LREAL#0.0, LREAL#0.0, LREAL#0.0, LREAL#0.0, LREAL#0.0, LREAL#19.579149162561258, LREAL#19.593929605703352, LREAL#19.608190954002232, LREAL#19.62195143826828, LREAL#19.635228649038805, LREAL#19.648039559064692, LREAL#19.660400545007292, LREAL#19.672327408373313, LREAL#19.683835395714475, LREAL#19.694939218117742, LREAL#19.705653070011053, LREAL#19.715990647308583, LREAL#19.725965164918737, LREAL#19.735589373637257, LREAL#19.74487557644704, LREAL#19.753835644245491, LREAL#19.762481031019547, LREAL#19.77082278848771, LREAL#19.778871580227889, LREAL#19.786637695309036, LREAL#19.794131061444048, LREAL#19.801361257680728, LREAL#19.808337526647041, LREAL#19.815068786366307, LREAL#19.821563641657438, LREAL#19.827830395134797, LREAL#19.833877057821745, LREAL#19.839711359391419, LREAL#19.845340758047868, LREAL#19.850772450060148, LREAL#19.856013378961581, LREAL#19.861070244425928, LREAL#19.865949510831836, LREAL#19.870657415526487, LREAL#19.875199976799031, LREAL#19.879583001573998, LREAL#19.883812092834489, LREAL#19.88789265678469, LREAL#19.891829909760816, LREAL#19.895628884899349, LREAL#19.899294438571086, LREAL#19.902831256589216, LREAL#0.0, LREAL#0.0, LREAL#0.0, LREAL#0.0, LREAL#0.0, LREAL#0.0, LREAL#0.0, LREAL#0.0, LREAL#19.593929605703352, LREAL#19.608190954002232, LREAL#19.62195143826828, LREAL#19.635228649038805, LREAL#19.648039559064692, LREAL#19.660400545007292, LREAL#19.672327408373313, LREAL#19.683835395714475, LREAL#19.694939218117742, LREAL#19.705653070011053, LREAL#19.715990647308583, LREAL#19.725965164918737, LREAL#19.735589373637257, LREAL#19.74487557644704, LREAL#19.753835644245491, LREAL#19.762481031019547, LREAL#19.77082278848771, LREAL#19.778871580227889, LREAL#19.786637695309036, LREAL#19.794131061444048, LREAL#19.801361257680728, LREAL#19.808337526647041, LREAL#19.815068786366307, LREAL#19.821563641657438, LREAL#19.827830395134797, LREAL#19.833877057821745, LREAL#19.839711359391419, LREAL#19.845340758047868, LREAL#19.850772450060148, LREAL#19.856013378961581, LREAL#19.861070244425928, LREAL#19.865949510831836, LREAL#19.870657415526487, LREAL#19.875199976799031, LREAL#19.879583001573998, LREAL#19.883812092834489, LREAL#19.88789265678469, LREAL#19.891829909760816, LREAL#19.895628884899349, LREAL#19.899294438571086, LREAL#19.902831256589216, LREAL#0.0, LREAL#0.0, LREAL#0.0, LREAL#0.0, LREAL#0.0, LREAL#0.0, LREAL#0.0, LREAL#0.0, LREAL#0.0, LREAL#19.608190954002232, LREAL#19.62195143826828, LREAL#19.635228649038805, LREAL#19.648039559064692, LREAL#19.660400545007292, LREAL#19.672327408373313, LREAL#19.683835395714475, LREAL#19.694939218117742, LREAL#19.705653070011053, LREAL#19.715990647308583, LREAL#19.725965164918737, LREAL#19.735589373637257, LREAL#19.74487557644704, LREAL#19.753835644245491, LREAL#19.762481031019547, LREAL#19.77082278848771, LREAL#19.778871580227889, LREAL#19.786637695309036, LREAL#19.794131061444048, LREAL#19.801361257680728, LREAL#19.808337526647041, LREAL#19.815068786366307, LREAL#19.821563641657438, LREAL#19.827830395134797, LREAL#19.833877057821745, LREAL#19.839711359391419, LREAL#19.845340758047868, LREAL#19.850772450060148, LREAL#19.856013378961581, LREAL#19.861070244425928, LREAL#19.865949510831836, LREAL#19.870657415526487, LREAL#19.875199976799031, LREAL#19.879583001573998, LREAL#19.883812092834489, LREAL#19.88789265678469, LREAL#19.891829909760816, LREAL#19.895628884899349, LREAL#19.899294438571086, LREAL#19.902831256589216, LREAL#0.0, LREAL#0.0, LREAL#0.0, LREAL#0.0, LREAL#0.0, LREAL#0.0, LREAL#0.0, LREAL#0.0, LREAL#0.0, LREAL#0.0, LREAL#19.62195143826828, LREAL#19.635228649038805, LREAL#19.648039559064692, LREAL#19.660400545007292, LREAL#19.672327408373313, LREAL#19.683835395714475, LREAL#19.694939218117742, LREAL#19.705653070011053, LREAL#19.715990647308583, LREAL#19.725965164918737, LREAL#19.735589373637257, LREAL#19.74487557644704, LREAL#19.753835644245491, LREAL#19.762481031019547, LREAL#19.77082278848771, LREAL#19.778871580227889, LREAL#19.786637695309036, LREAL#19.794131061444048, LREAL#19.801361257680728, LREAL#19.808337526647041, LREAL#19.815068786366307, LREAL#19.821563641657438, LREAL#19.827830395134797, LREAL#19.833877057821745, LREAL#19.839711359391419, LREAL#19.845340758047868, LREAL#19.850772450060148, LREAL#19.856013378961581, LREAL#19.861070244425928, LREAL#19.865949510831836, LREAL#19.870657415526487, LREAL#19.875199976799031, LREAL#19.879583001573998, LREAL#19.883812092834489, LREAL#19.88789265678469, LREAL#19.891829909760816, LREAL#19.895628884899349, LREAL#19.899294438571086, LREAL#19.902831256589216, LREAL#0.0, LREAL#0.0, LREAL#0.0, LREAL#0.0, LREAL#0.0, LREAL#0.0, LREAL#0.0, LREAL#0.0, LREAL#0.0, LREAL#0.0, LREAL#0.0, LREAL#19.635228649038805, LREAL#19.648039559064692, LREAL#19.660400545007292, LREAL#19.672327408373313, LREAL#19.683835395714475, LREAL#19.694939218117742, LREAL#19.705653070011053, LREAL#19.715990647308583, LREAL#19.725965164918737, LREAL#19.735589373637257, LREAL#19.74487557644704, LREAL#19.753835644245491, LREAL#19.762481031019547, LREAL#19.77082278848771, LREAL#19.778871580227889, LREAL#19.786637695309036, LREAL#19.794131061444048, LREAL#19.801361257680728, LREAL#19.808337526647041, LREAL#19.815068786366307, LREAL#19.821563641657438, LREAL#19.827830395134797, LREAL#19.833877057821745, LREAL#19.839711359391419, LREAL#19.845340758047868, LREAL#19.850772450060148, LREAL#19.856013378961581, LREAL#19.861070244425928, LREAL#19.865949510831836, LREAL#19.870657415526487, LREAL#19.875199976799031, LREAL#19.879583001573998, LREAL#19.883812092834489, LREAL#19.88789265678469, LREAL#19.891829909760816, LREAL#19.895628884899349, LREAL#19.899294438571086, LREAL#19.902831256589216, LREAL#0.0, LREAL#0.0, LREAL#0.0, LREAL#0.0, LREAL#0.0, LREAL#0.0, LREAL#0.0, LREAL#0.0, LREAL#0.0, LREAL#0.0, LREAL#0.0, LREAL#0.0, LREAL#19.648039559064692, LREAL#19.660400545007292, LREAL#19.672327408373313, LREAL#19.683835395714475, LREAL#19.694939218117742, LREAL#19.705653070011053, LREAL#19.715990647308583, LREAL#19.725965164918737, LREAL#19.735589373637257, LREAL#19.74487557644704, LREAL#19.753835644245491, LREAL#19.762481031019547, LREAL#19.77082278848771, LREAL#19.778871580227889, LREAL#19.786637695309036, LREAL#19.794131061444048, LREAL#19.801361257680728, LREAL#19.808337526647041, LREAL#19.815068786366307, LREAL#19.821563641657438, LREAL#19.827830395134797, LREAL#19.833877057821745, LREAL#19.839711359391419, LREAL#19.845340758047868, LREAL#19.850772450060148, LREAL#19.856013378961581, LREAL#19.861070244425928, LREAL#19.865949510831836, LREAL#19.870657415526487, LREAL#19.875199976799031, LREAL#19.879583001573998, LREAL#19.883812092834489, LREAL#19.88789265678469, LREAL#19.891829909760816, LREAL#19.895628884899349, LREAL#19.899294438571086, LREAL#19.902831256589216, LREAL#0.0, LREAL#0.0, LREAL#0.0, LREAL#0.0, LREAL#0.0, LREAL#0.0, LREAL#0.0, LREAL#0.0, LREAL#0.0, LREAL#0.0, LREAL#0.0, LREAL#0.0, LREAL#0.0, LREAL#19.660400545007292, LREAL#19.672327408373313, LREAL#19.683835395714475, LREAL#19.694939218117742, LREAL#19.705653070011053, LREAL#19.715990647308583, LREAL#19.725965164918737, LREAL#19.735589373637257, LREAL#19.74487557644704, LREAL#19.753835644245491, LREAL#19.762481031019547, LREAL#19.77082278848771, LREAL#19.778871580227889, LREAL#19.786637695309036, LREAL#19.794131061444048, LREAL#19.801361257680728, LREAL#19.808337526647041, LREAL#19.815068786366307, LREAL#19.821563641657438, LREAL#19.827830395134797, LREAL#19.833877057821745, LREAL#19.839711359391419, LREAL#19.845340758047868, LREAL#19.850772450060148, LREAL#19.856013378961581, LREAL#19.861070244425928, LREAL#19.865949510831836, LREAL#19.870657415526487, LREAL#19.875199976799031, LREAL#19.879583001573998, LREAL#19.883812092834489, LREAL#19.88789265678469, LREAL#19.891829909760816, LREAL#19.895628884899349, LREAL#19.899294438571086, LREAL#19.902831256589216, LREAL#0.0, LREAL#0.0, LREAL#0.0, LREAL#0.0, LREAL#0.0, LREAL#0.0, LREAL#0.0, LREAL#0.0, LREAL#0.0, LREAL#0.0, LREAL#0.0, LREAL#0.0, LREAL#0.0, LREAL#0.0, LREAL#19.672327408373313, LREAL#19.683835395714475, LREAL#19.694939218117742, LREAL#19.705653070011053, LREAL#19.715990647308583, LREAL#19.725965164918737, LREAL#19.735589373637257, LREAL#19.74487557644704, LREAL#19.753835644245491, LREAL#19.762481031019547, LREAL#19.77082278848771, LREAL#19.778871580227889, LREAL#19.786637695309036, LREAL#19.794131061444048, LREAL#19.801361257680728, LREAL#19.808337526647041, LREAL#19.815068786366307, LREAL#19.821563641657438, LREAL#19.827830395134797, LREAL#19.833877057821745, LREAL#19.839711359391419, LREAL#19.845340758047868, LREAL#19.850772450060148, LREAL#19.856013378961581, LREAL#19.861070244425928, LREAL#19.865949510831836, LREAL#19.870657415526487, LREAL#19.875199976799031, LREAL#19.879583001573998, LREAL#19.883812092834489, LREAL#19.88789265678469, LREAL#19.891829909760816, LREAL#19.895628884899349, LREAL#19.899294438571086, LREAL#19.902831256589216, LREAL#0.0, LREAL#0.0, LREAL#0.0, LREAL#0.0, LREAL#0.0, LREAL#0.0, LREAL#0.0, LREAL#0.0, LREAL#0.0, LREAL#0.0, LREAL#0.0, LREAL#0.0, LREAL#0.0, LREAL#0.0, LREAL#0.0, LREAL#19.683835395714475, LREAL#19.694939218117742, LREAL#19.705653070011053, LREAL#19.715990647308583, LREAL#19.725965164918737, LREAL#19.735589373637257, LREAL#19.74487557644704, LREAL#19.753835644245491, LREAL#19.762481031019547, LREAL#19.77082278848771, LREAL#19.778871580227889, LREAL#19.786637695309036, LREAL#19.794131061444048, LREAL#19.801361257680728, LREAL#19.808337526647041, LREAL#19.815068786366307, LREAL#19.821563641657438, LREAL#19.827830395134797, LREAL#19.833877057821745, LREAL#19.839711359391419, LREAL#19.845340758047868, LREAL#19.850772450060148, LREAL#19.856013378961581, LREAL#19.861070244425928, LREAL#19.865949510831836, LREAL#19.870657415526487, LREAL#19.875199976799031, LREAL#19.879583001573998, LREAL#19.883812092834489, LREAL#19.88789265678469, LREAL#19.891829909760816, LREAL#19.895628884899349, LREAL#19.899294438571086, LREAL#19.902831256589216, LREAL#0.0, LREAL#0.0, LREAL#0.0, LREAL#0.0, LREAL#0.0, LREAL#0.0, LREAL#0.0, LREAL#0.0, LREAL#0.0, LREAL#0.0, LREAL#0.0, LREAL#0.0, LREAL#0.0, LREAL#0.0, LREAL#0.0, LREAL#0.0, LREAL#19.694939218117742, LREAL#19.705653070011053, LREAL#19.715990647308583, LREAL#19.725965164918737, LREAL#19.735589373637257, LREAL#19.74487557644704, LREAL#19.753835644245491, LREAL#19.762481031019547, LREAL#19.77082278848771, LREAL#19.778871580227889, LREAL#19.786637695309036, LREAL#19.794131061444048, LREAL#19.801361257680728, LREAL#19.808337526647041, LREAL#19.815068786366307, LREAL#19.821563641657438, LREAL#19.827830395134797, LREAL#19.833877057821745, LREAL#19.839711359391419, LREAL#19.845340758047868, LREAL#19.850772450060148, LREAL#19.856013378961581, LREAL#19.861070244425928, LREAL#19.865949510831836, LREAL#19.870657415526487, LREAL#19.875199976799031, LREAL#19.879583001573998, LREAL#19.883812092834489, LREAL#19.88789265678469, LREAL#19.891829909760816, LREAL#19.895628884899349, LREAL#19.899294438571086, LREAL#19.902831256589216, LREAL#0.0, LREAL#0.0, LREAL#0.0, LREAL#0.0, LREAL#0.0, LREAL#0.0, LREAL#0.0, LREAL#0.0, LREAL#0.0, LREAL#0.0, LREAL#0.0, LREAL#0.0, LREAL#0.0, LREAL#0.0, LREAL#0.0, LREAL#0.0, LREAL#0.0, LREAL#19.705653070011053, LREAL#19.715990647308583, LREAL#19.725965164918737, LREAL#19.735589373637257, LREAL#19.74487557644704, LREAL#19.753835644245491, LREAL#19.762481031019547, LREAL#19.77082278848771, LREAL#19.778871580227889, LREAL#19.786637695309036, LREAL#19.794131061444048, LREAL#19.801361257680728, LREAL#19.808337526647041, LREAL#19.815068786366307, LREAL#19.821563641657438, LREAL#19.827830395134797, LREAL#19.833877057821745, LREAL#19.839711359391419, LREAL#19.845340758047868, LREAL#19.850772450060148, LREAL#19.856013378961581, LREAL#19.861070244425928, LREAL#19.865949510831836, LREAL#19.870657415526487, LREAL#19.875199976799031, LREAL#19.879583001573998, LREAL#19.883812092834489, LREAL#19.88789265678469, LREAL#19.891829909760816, LREAL#19.895628884899349, LREAL#19.899294438571086, LREAL#19.902831256589216, LREAL#0.0, LREAL#0.0, LREAL#0.0, LREAL#0.0, LREAL#0.0, LREAL#0.0, LREAL#0.0, LREAL#0.0, LREAL#0.0, LREAL#0.0, LREAL#0.0, LREAL#0.0, LREAL#0.0, LREAL#0.0, LREAL#0.0, LREAL#0.0, LREAL#0.0, LREAL#0.0, LREAL#19.715990647308583, LREAL#19.725965164918737, LREAL#19.735589373637257, LREAL#19.74487557644704, LREAL#19.753835644245491, LREAL#19.762481031019547, LREAL#19.77082278848771, LREAL#19.778871580227889, LREAL#19.786637695309036, LREAL#19.794131061444048, LREAL#19.801361257680728, LREAL#19.808337526647041, LREAL#19.815068786366307, LREAL#19.821563641657438, LREAL#19.827830395134797, LREAL#19.833877057821745, LREAL#19.839711359391419, LREAL#19.845340758047868, LREAL#19.850772450060148, LREAL#19.856013378961581, LREAL#19.861070244425928, LREAL#19.865949510831836, LREAL#19.870657415526487, LREAL#19.875199976799031, LREAL#19.879583001573998, LREAL#19.883812092834489, LREAL#19.88789265678469, LREAL#19.891829909760816, LREAL#19.895628884899349, LREAL#19.899294438571086, LREAL#19.902831256589216, LREAL#0.0, LREAL#0.0, LREAL#0.0, LREAL#0.0, LREAL#0.0, LREAL#0.0, LREAL#0.0, LREAL#0.0, LREAL#0.0, LREAL#0.0, LREAL#0.0, LREAL#0.0, LREAL#0.0, LREAL#0.0, LREAL#0.0, LREAL#0.0, LREAL#0.0, LREAL#0.0, LREAL#0.0, LREAL#19.725965164918737, LREAL#19.735589373637257, LREAL#19.74487557644704, LREAL#19.753835644245491, LREAL#19.762481031019547, LREAL#19.77082278848771, LREAL#19.778871580227889, LREAL#19.786637695309036, LREAL#19.794131061444048, LREAL#19.801361257680728, LREAL#19.808337526647041, LREAL#19.815068786366307, LREAL#19.821563641657438, LREAL#19.827830395134797, LREAL#19.833877057821745, LREAL#19.839711359391419, LREAL#19.845340758047868, LREAL#19.850772450060148, LREAL#19.856013378961581, LREAL#19.861070244425928, LREAL#19.865949510831836, LREAL#19.870657415526487, LREAL#19.875199976799031, LREAL#19.879583001573998, LREAL#19.883812092834489, LREAL#19.88789265678469, LREAL#19.891829909760816, LREAL#19.895628884899349, LREAL#19.899294438571086, LREAL#19.902831256589216, LREAL#0.0, LREAL#0.0, LREAL#0.0, LREAL#0.0, LREAL#0.0, LREAL#0.0, LREAL#0.0, LREAL#0.0, LREAL#0.0, LREAL#0.0, LREAL#0.0, LREAL#0.0, LREAL#0.0, LREAL#0.0, LREAL#0.0, LREAL#0.0, LREAL#0.0, LREAL#0.0, LREAL#0.0, LREAL#0.0, LREAL#19.735589373637257, LREAL#19.74487557644704, LREAL#19.753835644245491, LREAL#19.762481031019547, LREAL#19.77082278848771, LREAL#19.778871580227889, LREAL#19.786637695309036, LREAL#19.794131061444048, LREAL#19.801361257680728, LREAL#19.808337526647041, LREAL#19.815068786366307, LREAL#19.821563641657438, LREAL#19.827830395134797, LREAL#19.833877057821745, LREAL#19.839711359391419, LREAL#19.845340758047868, LREAL#19.850772450060148, LREAL#19.856013378961581, LREAL#19.861070244425928, LREAL#19.865949510831836, LREAL#19.870657415526487, LREAL#19.875199976799031, LREAL#19.879583001573998, LREAL#19.883812092834489, LREAL#19.88789265678469, LREAL#19.891829909760816, LREAL#19.895628884899349, LREAL#19.899294438571086, LREAL#19.902831256589216, LREAL#0.0, LREAL#0.0, LREAL#0.0, LREAL#0.0, LREAL#0.0, LREAL#0.0, LREAL#0.0, LREAL#0.0, LREAL#0.0, LREAL#0.0, LREAL#0.0, LREAL#0.0, LREAL#0.0, LREAL#0.0, LREAL#0.0, LREAL#0.0, LREAL#0.0, LREAL#0.0, LREAL#0.0, LREAL#0.0, LREAL#0.0, LREAL#19.74487557644704, LREAL#19.753835644245491, LREAL#19.762481031019547, LREAL#19.77082278848771, LREAL#19.778871580227889, LREAL#19.786637695309036, LREAL#19.794131061444048, LREAL#19.801361257680728, LREAL#19.808337526647041, LREAL#19.815068786366307, LREAL#19.821563641657438, LREAL#19.827830395134797, LREAL#19.833877057821745, LREAL#19.839711359391419, LREAL#19.845340758047868, LREAL#19.850772450060148, LREAL#19.856013378961581, LREAL#19.861070244425928, LREAL#19.865949510831836, LREAL#19.870657415526487, LREAL#19.875199976799031, LREAL#19.879583001573998, LREAL#19.883812092834489, LREAL#19.88789265678469, LREAL#19.891829909760816, LREAL#19.895628884899349, LREAL#19.899294438571086, LREAL#19.902831256589216, LREAL#0.0, LREAL#0.0, LREAL#0.0, LREAL#0.0, LREAL#0.0, LREAL#0.0, LREAL#0.0, LREAL#0.0, LREAL#0.0, LREAL#0.0, LREAL#0.0, LREAL#0.0, LREAL#0.0, LREAL#0.0, LREAL#0.0, LREAL#0.0, LREAL#0.0, LREAL#0.0, LREAL#0.0, LREAL#0.0, LREAL#0.0, LREAL#0.0, LREAL#19.753835644245491, LREAL#19.762481031019547, LREAL#19.77082278848771, LREAL#19.778871580227889, LREAL#19.786637695309036, LREAL#19.794131061444048, LREAL#19.801361257680728, LREAL#19.808337526647041, LREAL#19.815068786366307, LREAL#19.821563641657438, LREAL#19.827830395134797, LREAL#19.833877057821745, LREAL#19.839711359391419, LREAL#19.845340758047868, LREAL#19.850772450060148, LREAL#19.856013378961581, LREAL#19.861070244425928, LREAL#19.865949510831836, LREAL#19.870657415526487, LREAL#19.875199976799031, LREAL#19.879583001573998, LREAL#19.883812092834489, LREAL#19.88789265678469, LREAL#19.891829909760816, LREAL#19.895628884899349, LREAL#19.899294438571086, LREAL#19.902831256589216, LREAL#0.0, LREAL#0.0, LREAL#0.0, LREAL#0.0, LREAL#0.0, LREAL#0.0, LREAL#0.0, LREAL#0.0, LREAL#0.0, LREAL#0.0, LREAL#0.0, LREAL#0.0, LREAL#0.0, LREAL#0.0, LREAL#0.0, LREAL#0.0, LREAL#0.0, LREAL#0.0, LREAL#0.0, LREAL#0.0, LREAL#0.0, LREAL#0.0, LREAL#0.0, LREAL#19.762481031019547, LREAL#19.77082278848771, LREAL#19.778871580227889, LREAL#19.786637695309036, LREAL#19.794131061444048, LREAL#19.801361257680728, LREAL#19.808337526647041, LREAL#19.815068786366307, LREAL#19.821563641657438, LREAL#19.827830395134797, LREAL#19.833877057821745, LREAL#19.839711359391419, LREAL#19.845340758047868, LREAL#19.850772450060148, LREAL#19.856013378961581, LREAL#19.861070244425928, LREAL#19.865949510831836, LREAL#19.870657415526487, LREAL#19.875199976799031, LREAL#19.879583001573998, LREAL#19.883812092834489, LREAL#19.88789265678469, LREAL#19.891829909760816, LREAL#19.895628884899349, LREAL#19.899294438571086, LREAL#19.902831256589216, LREAL#0.0, LREAL#0.0, LREAL#0.0, LREAL#0.0, LREAL#0.0, LREAL#0.0, LREAL#0.0, LREAL#0.0, LREAL#0.0, LREAL#0.0, LREAL#0.0, LREAL#0.0, LREAL#0.0, LREAL#0.0, LREAL#0.0, LREAL#0.0, LREAL#0.0, LREAL#0.0, LREAL#0.0, LREAL#0.0, LREAL#0.0, LREAL#0.0, LREAL#0.0, LREAL#0.0, LREAL#19.77082278848771, LREAL#19.778871580227889, LREAL#19.786637695309036, LREAL#19.794131061444048, LREAL#19.801361257680728, LREAL#19.808337526647041, LREAL#19.815068786366307, LREAL#19.821563641657438, LREAL#19.827830395134797, LREAL#19.833877057821745, LREAL#19.839711359391419, LREAL#19.845340758047868, LREAL#19.850772450060148, LREAL#19.856013378961581, LREAL#19.861070244425928, LREAL#19.865949510831836, LREAL#19.870657415526487, LREAL#19.875199976799031, LREAL#19.879583001573998, LREAL#19.883812092834489, LREAL#19.88789265678469, LREAL#19.891829909760816, LREAL#19.895628884899349, LREAL#19.899294438571086, LREAL#19.902831256589216, LREAL#0.0, LREAL#0.0, LREAL#0.0, LREAL#0.0, LREAL#0.0, LREAL#0.0, LREAL#0.0, LREAL#0.0, LREAL#0.0, LREAL#0.0, LREAL#0.0, LREAL#0.0, LREAL#0.0, LREAL#0.0, LREAL#0.0, LREAL#0.0, LREAL#0.0, LREAL#0.0, LREAL#0.0, LREAL#0.0, LREAL#0.0, LREAL#0.0, LREAL#0.0, LREAL#0.0, LREAL#0.0, LREAL#19.778871580227889, LREAL#19.786637695309036, LREAL#19.794131061444048, LREAL#19.801361257680728, LREAL#19.808337526647041, LREAL#19.815068786366307, LREAL#19.821563641657438, LREAL#19.827830395134797, LREAL#19.833877057821745, LREAL#19.839711359391419, LREAL#19.845340758047868, LREAL#19.850772450060148, LREAL#19.856013378961581, LREAL#19.861070244425928, LREAL#19.865949510831836, LREAL#19.870657415526487, LREAL#19.875199976799031, LREAL#19.879583001573998, LREAL#19.883812092834489, LREAL#19.88789265678469, LREAL#19.891829909760816, LREAL#19.895628884899349, LREAL#19.899294438571086, LREAL#19.902831256589216, LREAL#0.0, LREAL#0.0, LREAL#0.0, LREAL#0.0, LREAL#0.0, LREAL#0.0, LREAL#0.0, LREAL#0.0, LREAL#0.0, LREAL#0.0, LREAL#0.0, LREAL#0.0, LREAL#0.0, LREAL#0.0, LREAL#0.0, LREAL#0.0, LREAL#0.0, LREAL#0.0, LREAL#0.0, LREAL#0.0, LREAL#0.0, LREAL#0.0, LREAL#0.0, LREAL#0.0, LREAL#0.0, LREAL#0.0, LREAL#19.786637695309036, LREAL#19.794131061444048, LREAL#19.801361257680728, LREAL#19.808337526647041, LREAL#19.815068786366307, LREAL#19.821563641657438, LREAL#19.827830395134797, LREAL#19.833877057821745, LREAL#19.839711359391419, LREAL#19.845340758047868, LREAL#19.850772450060148, LREAL#19.856013378961581, LREAL#19.861070244425928, LREAL#19.865949510831836, LREAL#19.870657415526487, LREAL#19.875199976799031, LREAL#19.879583001573998, LREAL#19.883812092834489, LREAL#19.88789265678469, LREAL#19.891829909760816, LREAL#19.895628884899349, LREAL#19.899294438571086, LREAL#19.902831256589216, LREAL#0.0, LREAL#0.0, LREAL#0.0, LREAL#0.0, LREAL#0.0, LREAL#0.0, LREAL#0.0, LREAL#0.0, LREAL#0.0, LREAL#0.0, LREAL#0.0, LREAL#0.0, LREAL#0.0, LREAL#0.0, LREAL#0.0, LREAL#0.0, LREAL#0.0, LREAL#0.0, LREAL#0.0, LREAL#0.0, LREAL#0.0, LREAL#0.0, LREAL#0.0, LREAL#0.0, LREAL#0.0, LREAL#0.0, LREAL#0.0, LREAL#19.794131061444048, LREAL#19.801361257680728, LREAL#19.808337526647041, LREAL#19.815068786366307, LREAL#19.821563641657438, LREAL#19.827830395134797, LREAL#19.833877057821745, LREAL#19.839711359391419, LREAL#19.845340758047868, LREAL#19.850772450060148, LREAL#19.856013378961581, LREAL#19.861070244425928, LREAL#19.865949510831836, LREAL#19.870657415526487, LREAL#19.875199976799031, LREAL#19.879583001573998, LREAL#19.883812092834489, LREAL#19.88789265678469, LREAL#19.891829909760816, LREAL#19.895628884899349, LREAL#19.899294438571086, LREAL#19.902831256589216, LREAL#0.0, LREAL#0.0, LREAL#0.0, LREAL#0.0, LREAL#0.0, LREAL#0.0, LREAL#0.0, LREAL#0.0, LREAL#0.0, LREAL#0.0, LREAL#0.0, LREAL#0.0, LREAL#0.0, LREAL#0.0, LREAL#0.0, LREAL#0.0, LREAL#0.0, LREAL#0.0, LREAL#0.0, LREAL#0.0, LREAL#0.0, LREAL#0.0, LREAL#0.0, LREAL#0.0, LREAL#0.0, LREAL#0.0, LREAL#0.0, LREAL#0.0, LREAL#19.801361257680728, LREAL#19.808337526647041, LREAL#19.815068786366307, LREAL#19.821563641657438, LREAL#19.827830395134797, LREAL#19.833877057821745, LREAL#19.839711359391419, LREAL#19.845340758047868, LREAL#19.850772450060148, LREAL#19.856013378961581, LREAL#19.861070244425928, LREAL#19.865949510831836, LREAL#19.870657415526487, LREAL#19.875199976799031, LREAL#19.879583001573998, LREAL#19.883812092834489, LREAL#19.88789265678469, LREAL#19.891829909760816, LREAL#19.895628884899349, LREAL#19.899294438571086, LREAL#19.902831256589216, LREAL#0.0, LREAL#0.0, LREAL#0.0, LREAL#0.0, LREAL#0.0, LREAL#0.0, LREAL#0.0, LREAL#0.0, LREAL#0.0, LREAL#0.0, LREAL#0.0, LREAL#0.0, LREAL#0.0, LREAL#0.0, LREAL#0.0, LREAL#0.0, LREAL#0.0, LREAL#0.0, LREAL#0.0, LREAL#0.0, LREAL#0.0, LREAL#0.0, LREAL#0.0, LREAL#0.0, LREAL#0.0, LREAL#0.0, LREAL#0.0, LREAL#0.0, LREAL#0.0, LREAL#19.808337526647041, LREAL#19.815068786366307, LREAL#19.821563641657438, LREAL#19.827830395134797, LREAL#19.833877057821745, LREAL#19.839711359391419, LREAL#19.845340758047868, LREAL#19.850772450060148, LREAL#19.856013378961581, LREAL#19.861070244425928, LREAL#19.865949510831836, LREAL#19.870657415526487, LREAL#19.875199976799031, LREAL#19.879583001573998, LREAL#19.883812092834489, LREAL#19.88789265678469, LREAL#19.891829909760816, LREAL#19.895628884899349, LREAL#19.899294438571086, LREAL#19.902831256589216, LREAL#0.0, LREAL#0.0, LREAL#0.0, LREAL#0.0, LREAL#0.0, LREAL#0.0, LREAL#0.0, LREAL#0.0, LREAL#0.0, LREAL#0.0, LREAL#0.0, LREAL#0.0, LREAL#0.0, LREAL#0.0, LREAL#0.0, LREAL#0.0, LREAL#0.0, LREAL#0.0, LREAL#0.0, LREAL#0.0, LREAL#0.0, LREAL#0.0, LREAL#0.0, LREAL#0.0, LREAL#0.0, LREAL#0.0, LREAL#0.0, LREAL#0.0, LREAL#0.0, LREAL#0.0, LREAL#19.815068786366307, LREAL#19.821563641657438, LREAL#19.827830395134797, LREAL#19.833877057821745, LREAL#19.839711359391419, LREAL#19.845340758047868, LREAL#19.850772450060148, LREAL#19.856013378961581, LREAL#19.861070244425928, LREAL#19.865949510831836, LREAL#19.870657415526487, LREAL#19.875199976799031, LREAL#19.879583001573998, LREAL#19.883812092834489, LREAL#19.88789265678469, LREAL#19.891829909760816, LREAL#19.895628884899349, LREAL#19.899294438571086, LREAL#19.902831256589216, LREAL#0.0, LREAL#0.0, LREAL#0.0, LREAL#0.0, LREAL#0.0, LREAL#0.0, LREAL#0.0, LREAL#0.0, LREAL#0.0, LREAL#0.0, LREAL#0.0, LREAL#0.0, LREAL#0.0, LREAL#0.0, LREAL#0.0, LREAL#0.0, LREAL#0.0, LREAL#0.0, LREAL#0.0, LREAL#0.0, LREAL#0.0, LREAL#0.0, LREAL#0.0, LREAL#0.0, LREAL#0.0, LREAL#0.0, LREAL#0.0, LREAL#0.0, LREAL#0.0, LREAL#0.0, LREAL#0.0, LREAL#19.821563641657438, LREAL#19.827830395134797, LREAL#19.833877057821745, LREAL#19.839711359391419, LREAL#19.845340758047868, LREAL#19.850772450060148, LREAL#19.856013378961581, LREAL#19.861070244425928, LREAL#19.865949510831836, LREAL#19.870657415526487, LREAL#19.875199976799031, LREAL#19.879583001573998, LREAL#19.883812092834489, LREAL#19.88789265678469, LREAL#19.891829909760816, LREAL#19.895628884899349, LREAL#19.899294438571086, LREAL#19.902831256589216, LREAL#0.0, LREAL#0.0, LREAL#0.0, LREAL#0.0, LREAL#0.0, LREAL#0.0, LREAL#0.0, LREAL#0.0, LREAL#0.0, LREAL#0.0, LREAL#0.0, LREAL#0.0, LREAL#0.0, LREAL#0.0, LREAL#0.0, LREAL#0.0, LREAL#0.0, LREAL#0.0, LREAL#0.0, LREAL#0.0, LREAL#0.0, LREAL#0.0, LREAL#0.0, LREAL#0.0, LREAL#0.0, LREAL#0.0, LREAL#0.0, LREAL#0.0, LREAL#0.0, LREAL#0.0, LREAL#0.0, LREAL#0.0, LREAL#19.827830395134797, LREAL#19.833877057821745, LREAL#19.839711359391419, LREAL#19.845340758047868, LREAL#19.850772450060148, LREAL#19.856013378961581, LREAL#19.861070244425928, LREAL#19.865949510831836, LREAL#19.870657415526487, LREAL#19.875199976799031, LREAL#19.879583001573998, LREAL#19.883812092834489, LREAL#19.88789265678469, LREAL#19.891829909760816, LREAL#19.895628884899349, LREAL#19.899294438571086, LREAL#19.902831256589216, LREAL#0.0, LREAL#0.0, LREAL#0.0, LREAL#0.0, LREAL#0.0, LREAL#0.0, LREAL#0.0, LREAL#0.0, LREAL#0.0, LREAL#0.0, LREAL#0.0, LREAL#0.0, LREAL#0.0, LREAL#0.0, LREAL#0.0, LREAL#0.0, LREAL#0.0, LREAL#0.0, LREAL#0.0, LREAL#0.0, LREAL#0.0, LREAL#0.0, LREAL#0.0, LREAL#0.0, LREAL#0.0, LREAL#0.0, LREAL#0.0, LREAL#0.0, LREAL#0.0, LREAL#0.0, LREAL#0.0, LREAL#0.0, LREAL#0.0, LREAL#19.833877057821745, LREAL#19.839711359391419, LREAL#19.845340758047868, LREAL#19.850772450060148, LREAL#19.856013378961581, LREAL#19.861070244425928, LREAL#19.865949510831836, LREAL#19.870657415526487, LREAL#19.875199976799031, LREAL#19.879583001573998, LREAL#19.883812092834489, LREAL#19.88789265678469, LREAL#19.891829909760816, LREAL#19.895628884899349, LREAL#19.899294438571086, LREAL#19.902831256589216, LREAL#0.0, LREAL#0.0, LREAL#0.0, LREAL#0.0, LREAL#0.0, LREAL#0.0, LREAL#0.0, LREAL#0.0, LREAL#0.0, LREAL#0.0, LREAL#0.0, LREAL#0.0, LREAL#0.0, LREAL#0.0, LREAL#0.0, LREAL#0.0, LREAL#0.0, LREAL#0.0, LREAL#0.0, LREAL#0.0, LREAL#0.0, LREAL#0.0, LREAL#0.0, LREAL#0.0, LREAL#0.0, LREAL#0.0, LREAL#0.0, LREAL#0.0, LREAL#0.0, LREAL#0.0, LREAL#0.0, LREAL#0.0, LREAL#0.0, LREAL#0.0, LREAL#19.839711359391419, LREAL#19.845340758047868, LREAL#19.850772450060148, LREAL#19.856013378961581, LREAL#19.861070244425928, LREAL#19.865949510831836, LREAL#19.870657415526487, LREAL#19.875199976799031, LREAL#19.879583001573998, LREAL#19.883812092834489, LREAL#19.88789265678469, LREAL#19.891829909760816, LREAL#19.895628884899349, LREAL#19.899294438571086, LREAL#19.902831256589216, LREAL#0.0, LREAL#0.0, LREAL#0.0, LREAL#0.0, LREAL#0.0, LREAL#0.0, LREAL#0.0, LREAL#0.0, LREAL#0.0, LREAL#0.0, LREAL#0.0, LREAL#0.0, LREAL#0.0, LREAL#0.0, LREAL#0.0, LREAL#0.0, LREAL#0.0, LREAL#0.0, LREAL#0.0, LREAL#0.0, LREAL#0.0, LREAL#0.0, LREAL#0.0, LREAL#0.0, LREAL#0.0, LREAL#0.0, LREAL#0.0, LREAL#0.0, LREAL#0.0, LREAL#0.0, LREAL#0.0, LREAL#0.0, LREAL#0.0, LREAL#0.0, LREAL#0.0, LREAL#19.845340758047868, LREAL#19.850772450060148, LREAL#19.856013378961581, LREAL#19.861070244425928, LREAL#19.865949510831836, LREAL#19.870657415526487, LREAL#19.875199976799031, LREAL#19.879583001573998, LREAL#19.883812092834489, LREAL#19.88789265678469, LREAL#19.891829909760816, LREAL#19.895628884899349, LREAL#19.899294438571086, LREAL#19.902831256589216, LREAL#0.0, LREAL#0.0, LREAL#0.0, LREAL#0.0, LREAL#0.0, LREAL#0.0, LREAL#0.0, LREAL#0.0, LREAL#0.0, LREAL#0.0, LREAL#0.0, LREAL#0.0, LREAL#0.0, LREAL#0.0, LREAL#0.0, LREAL#0.0, LREAL#0.0, LREAL#0.0, LREAL#0.0, LREAL#0.0, LREAL#0.0, LREAL#0.0, LREAL#0.0, LREAL#0.0, LREAL#0.0, LREAL#0.0, LREAL#0.0, LREAL#0.0, LREAL#0.0, LREAL#0.0, LREAL#0.0, LREAL#0.0, LREAL#0.0, LREAL#0.0, LREAL#0.0, LREAL#0.0, LREAL#19.850772450060148, LREAL#19.856013378961581, LREAL#19.861070244425928, LREAL#19.865949510831836, LREAL#19.870657415526487, LREAL#19.875199976799031, LREAL#19.879583001573998, LREAL#19.883812092834489, LREAL#19.88789265678469, LREAL#19.891829909760816, LREAL#19.895628884899349, LREAL#19.899294438571086, LREAL#19.902831256589216, LREAL#0.0, LREAL#0.0, LREAL#0.0, LREAL#0.0, LREAL#0.0, LREAL#0.0, LREAL#0.0, LREAL#0.0, LREAL#0.0, LREAL#0.0, LREAL#0.0, LREAL#0.0, LREAL#0.0, LREAL#0.0, LREAL#0.0, LREAL#0.0, LREAL#0.0, LREAL#0.0, LREAL#0.0, LREAL#0.0, LREAL#0.0, LREAL#0.0, LREAL#0.0, LREAL#0.0, LREAL#0.0, LREAL#0.0, LREAL#0.0, LREAL#0.0, LREAL#0.0, LREAL#0.0, LREAL#0.0, LREAL#0.0, LREAL#0.0, LREAL#0.0, LREAL#0.0, LREAL#0.0, LREAL#0.0, LREAL#19.856013378961581, LREAL#19.861070244425928, LREAL#19.865949510831836, LREAL#19.870657415526487, LREAL#19.875199976799031, LREAL#19.879583001573998, LREAL#19.883812092834489, LREAL#19.88789265678469, LREAL#19.891829909760816, LREAL#19.895628884899349, LREAL#19.899294438571086, LREAL#19.902831256589216, LREAL#0.0, LREAL#0.0, LREAL#0.0, LREAL#0.0, LREAL#0.0, LREAL#0.0, LREAL#0.0, LREAL#0.0, LREAL#0.0, LREAL#0.0, LREAL#0.0, LREAL#0.0, LREAL#0.0, LREAL#0.0, LREAL#0.0, LREAL#0.0, LREAL#0.0, LREAL#0.0, LREAL#0.0, LREAL#0.0, LREAL#0.0, LREAL#0.0, LREAL#0.0, LREAL#0.0, LREAL#0.0, LREAL#0.0, LREAL#0.0, LREAL#0.0, LREAL#0.0, LREAL#0.0, LREAL#0.0, LREAL#0.0, LREAL#0.0, LREAL#0.0, LREAL#0.0, LREAL#0.0, LREAL#0.0, LREAL#0.0, LREAL#19.861070244425928, LREAL#19.865949510831836, LREAL#19.870657415526487, LREAL#19.875199976799031, LREAL#19.879583001573998, LREAL#19.883812092834489, LREAL#19.88789265678469, LREAL#19.891829909760816, LREAL#19.895628884899349, LREAL#19.899294438571086, LREAL#19.902831256589216, LREAL#0.0, LREAL#0.0, LREAL#0.0, LREAL#0.0, LREAL#0.0, LREAL#0.0, LREAL#0.0, LREAL#0.0, LREAL#0.0, LREAL#0.0, LREAL#0.0, LREAL#0.0, LREAL#0.0, LREAL#0.0, LREAL#0.0, LREAL#0.0, LREAL#0.0, LREAL#0.0, LREAL#0.0, LREAL#0.0, LREAL#0.0, LREAL#0.0, LREAL#0.0, LREAL#0.0, LREAL#0.0, LREAL#0.0, LREAL#0.0, LREAL#0.0, LREAL#0.0, LREAL#0.0, LREAL#0.0, LREAL#0.0, LREAL#0.0, LREAL#0.0, LREAL#0.0, LREAL#0.0, LREAL#0.0, LREAL#0.0, LREAL#0.0, LREAL#19.865949510831836, LREAL#19.870657415526487, LREAL#19.875199976799031, LREAL#19.879583001573998, LREAL#19.883812092834489, LREAL#19.88789265678469, LREAL#19.891829909760816, LREAL#19.895628884899349, LREAL#19.899294438571086, LREAL#19.902831256589216, LREAL#0.0, LREAL#0.0, LREAL#0.0, LREAL#0.0, LREAL#0.0, LREAL#0.0, LREAL#0.0, LREAL#0.0, LREAL#0.0, LREAL#0.0, LREAL#0.0, LREAL#0.0, LREAL#0.0, LREAL#0.0, LREAL#0.0, LREAL#0.0, LREAL#0.0, LREAL#0.0, LREAL#0.0, LREAL#0.0, LREAL#0.0, LREAL#0.0, LREAL#0.0, LREAL#0.0, LREAL#0.0, LREAL#0.0, LREAL#0.0, LREAL#0.0, LREAL#0.0, LREAL#0.0, LREAL#0.0, LREAL#0.0, LREAL#0.0, LREAL#0.0, LREAL#0.0, LREAL#0.0, LREAL#0.0, LREAL#0.0, LREAL#0.0, LREAL#0.0, LREAL#19.870657415526487, LREAL#19.875199976799031, LREAL#19.879583001573998, LREAL#19.883812092834489, LREAL#19.88789265678469, LREAL#19.891829909760816, LREAL#19.895628884899349, LREAL#19.899294438571086, LREAL#19.902831256589216, LREAL#0.0, LREAL#0.0, LREAL#0.0, LREAL#0.0, LREAL#0.0, LREAL#0.0, LREAL#0.0, LREAL#0.0, LREAL#0.0, LREAL#0.0, LREAL#0.0, LREAL#0.0, LREAL#0.0, LREAL#0.0, LREAL#0.0, LREAL#0.0, LREAL#0.0, LREAL#0.0, LREAL#0.0, LREAL#0.0, LREAL#0.0, LREAL#0.0, LREAL#0.0, LREAL#0.0, LREAL#0.0, LREAL#0.0, LREAL#0.0, LREAL#0.0, LREAL#0.0, LREAL#0.0, LREAL#0.0, LREAL#0.0, LREAL#0.0, LREAL#0.0, LREAL#0.0, LREAL#0.0, LREAL#0.0, LREAL#0.0, LREAL#0.0, LREAL#0.0, LREAL#0.0, LREAL#19.875199976799031, LREAL#19.879583001573998, LREAL#19.883812092834489, LREAL#19.88789265678469, LREAL#19.891829909760816, LREAL#19.895628884899349, LREAL#19.899294438571086, LREAL#19.902831256589216, LREAL#0.0, LREAL#0.0, LREAL#0.0, LREAL#0.0, LREAL#0.0, LREAL#0.0, LREAL#0.0, LREAL#0.0, LREAL#0.0, LREAL#0.0, LREAL#0.0, LREAL#0.0, LREAL#0.0, LREAL#0.0, LREAL#0.0, LREAL#0.0, LREAL#0.0, LREAL#0.0, LREAL#0.0, LREAL#0.0, LREAL#0.0, LREAL#0.0, LREAL#0.0, LREAL#0.0, LREAL#0.0, LREAL#0.0, LREAL#0.0, LREAL#0.0, LREAL#0.0, LREAL#0.0, LREAL#0.0, LREAL#0.0, LREAL#0.0, LREAL#0.0, LREAL#0.0, LREAL#0.0, LREAL#0.0, LREAL#0.0, LREAL#0.0, LREAL#0.0, LREAL#0.0, LREAL#0.0, LREAL#19.879583001573998, LREAL#19.883812092834489, LREAL#19.88789265678469, LREAL#19.891829909760816, LREAL#19.895628884899349, LREAL#19.899294438571086, LREAL#19.902831256589216, LREAL#0.0, LREAL#0.0, LREAL#0.0, LREAL#0.0, LREAL#0.0, LREAL#0.0, LREAL#0.0, LREAL#0.0, LREAL#0.0, LREAL#0.0, LREAL#0.0, LREAL#0.0, LREAL#0.0, LREAL#0.0, LREAL#0.0, LREAL#0.0, LREAL#0.0, LREAL#0.0, LREAL#0.0, LREAL#0.0, LREAL#0.0, LREAL#0.0, LREAL#0.0, LREAL#0.0, LREAL#0.0, LREAL#0.0, LREAL#0.0, LREAL#0.0, LREAL#0.0, LREAL#0.0, LREAL#0.0, LREAL#0.0, LREAL#0.0, LREAL#0.0, LREAL#0.0, LREAL#0.0, LREAL#0.0, LREAL#0.0, LREAL#0.0, LREAL#0.0, LREAL#0.0, LREAL#0.0, LREAL#0.0, LREAL#19.883812092834489, LREAL#19.88789265678469, LREAL#19.891829909760816, LREAL#19.895628884899349, LREAL#19.899294438571086, LREAL#19.902831256589216, LREAL#0.0, LREAL#0.0, LREAL#0.0, LREAL#0.0, LREAL#0.0, LREAL#0.0, LREAL#0.0, LREAL#0.0, LREAL#0.0, LREAL#0.0, LREAL#0.0, LREAL#0.0, LREAL#0.0, LREAL#0.0, LREAL#0.0, LREAL#0.0, LREAL#0.0, LREAL#0.0, LREAL#0.0, LREAL#0.0, LREAL#0.0, LREAL#0.0, LREAL#0.0, LREAL#0.0, LREAL#0.0, LREAL#0.0, LREAL#0.0, LREAL#0.0, LREAL#0.0, LREAL#0.0, LREAL#0.0, LREAL#0.0, LREAL#0.0, LREAL#0.0, LREAL#0.0, LREAL#0.0, LREAL#0.0, LREAL#0.0, LREAL#0.0, LREAL#0.0, LREAL#0.0, LREAL#0.0, LREAL#0.0, LREAL#0.0, LREAL#19.88789265678469, LREAL#19.891829909760816, LREAL#19.895628884899349, LREAL#19.899294438571086, LREAL#19.902831256589216, LREAL#0.0, LREAL#0.0, LREAL#0.0, LREAL#0.0, LREAL#0.0, LREAL#0.0, LREAL#0.0, LREAL#0.0, LREAL#0.0, LREAL#0.0, LREAL#0.0, LREAL#0.0, LREAL#0.0, LREAL#0.0, LREAL#0.0, LREAL#0.0, LREAL#0.0, LREAL#0.0, LREAL#0.0, LREAL#0.0, LREAL#0.0, LREAL#0.0, LREAL#0.0, LREAL#0.0, LREAL#0.0, LREAL#0.0, LREAL#0.0, LREAL#0.0, LREAL#0.0, LREAL#0.0, LREAL#0.0, LREAL#0.0, LREAL#0.0, LREAL#0.0, LREAL#0.0, LREAL#0.0, LREAL#0.0, LREAL#0.0, LREAL#0.0, LREAL#0.0, LREAL#0.0, LREAL#0.0, LREAL#0.0, LREAL#0.0, LREAL#0.0, LREAL#19.891829909760816, LREAL#19.895628884899349, LREAL#19.899294438571086, LREAL#19.902831256589216, LREAL#0.0, LREAL#0.0, LREAL#0.0, LREAL#0.0, LREAL#0.0, LREAL#0.0, LREAL#0.0, LREAL#0.0, LREAL#0.0, LREAL#0.0, LREAL#0.0, LREAL#0.0, LREAL#0.0, LREAL#0.0, LREAL#0.0, LREAL#0.0, LREAL#0.0, LREAL#0.0, LREAL#0.0, LREAL#0.0, LREAL#0.0, LREAL#0.0, LREAL#0.0, LREAL#0.0, LREAL#0.0, LREAL#0.0, LREAL#0.0, LREAL#0.0, LREAL#0.0, LREAL#0.0, LREAL#0.0, LREAL#0.0, LREAL#0.0, LREAL#0.0, LREAL#0.0, LREAL#0.0, LREAL#0.0, LREAL#0.0, LREAL#0.0, LREAL#0.0, LREAL#0.0, LREAL#0.0, LREAL#0.0, LREAL#0.0, LREAL#0.0, LREAL#0.0, LREAL#19.895628884899349, LREAL#19.899294438571086, LREAL#19.902831256589216, LREAL#0.0, LREAL#0.0, LREAL#0.0, LREAL#0.0, LREAL#0.0, LREAL#0.0, LREAL#0.0, LREAL#0.0, LREAL#0.0, LREAL#0.0, LREAL#0.0, LREAL#0.0, LREAL#0.0, LREAL#0.0, LREAL#0.0, LREAL#0.0, LREAL#0.0, LREAL#0.0, LREAL#0.0, LREAL#0.0, LREAL#0.0, LREAL#0.0, LREAL#0.0, LREAL#0.0, LREAL#0.0, LREAL#0.0, LREAL#0.0, LREAL#0.0, LREAL#0.0, LREAL#0.0, LREAL#0.0, LREAL#0.0, LREAL#0.0, LREAL#0.0, LREAL#0.0, LREAL#0.0, LREAL#0.0, LREAL#0.0, LREAL#0.0, LREAL#0.0, LREAL#0.0, LREAL#0.0, LREAL#0.0, LREAL#0.0, LREAL#0.0, LREAL#0.0, LREAL#0.0, LREAL#19.899294438571086, LREAL#19.902831256589216, LREAL#0.0, LREAL#0.0, LREAL#0.0, LREAL#0.0, LREAL#0.0, LREAL#0.0, LREAL#0.0, LREAL#0.0, LREAL#0.0, LREAL#0.0, LREAL#0.0, LREAL#0.0, LREAL#0.0, LREAL#0.0, LREAL#0.0, LREAL#0.0, LREAL#0.0, LREAL#0.0, LREAL#0.0, LREAL#0.0, LREAL#0.0, LREAL#0.0, LREAL#0.0, LREAL#0.0, LREAL#0.0, LREAL#0.0, LREAL#0.0, LREAL#0.0, LREAL#0.0, LREAL#0.0, LREAL#0.0, LREAL#0.0, LREAL#0.0, LREAL#0.0, LREAL#0.0, LREAL#0.0, LREAL#0.0, LREAL#0.0, LREAL#0.0, LREAL#0.0, LREAL#0.0, LREAL#0.0, LREAL#0.0, LREAL#0.0, LREAL#0.0, LREAL#0.0, LREAL#0.0, LREAL#0.0, LREAL#19.902831256589216, LREAL#0.0, LREAL#0.0, LREAL#0.0, LREAL#0.0, LREAL#0.0, LREAL#0.0, LREAL#0.0, LREAL#0.0, LREAL#0.0, LREAL#0.0, LREAL#0.0, LREAL#0.0, LREAL#0.0, LREAL#0.0, LREAL#0.0, LREAL#0.0, LREAL#0.0, LREAL#0.0, LREAL#0.0, LREAL#0.0, LREAL#0.0, LREAL#0.0, LREAL#0.0, LREAL#0.0, LREAL#0.0, LREAL#0.0, LREAL#0.0, LREAL#0.0, LREAL#0.0, LREAL#0.0, LREAL#0.0, LREAL#0.0, LREAL#0.0, LREAL#0.0, LREAL#0.0, LREAL#0.0, LREAL#0.0, LREAL#0.0, LREAL#0.0, LREAL#0.0, LREAL#0.0, LREAL#0.0, LREAL#0.0, LREAL#0.0, LREAL#0.0, LREAL#0.0, LREAL#0.0, LREAL#0.0, LREAL#0.0];
    Gain1_Gain : ARRAY[0..99] OF LREAL := [LREAL#0.0033971064571647839, LREAL#-0.0034147668244180235, LREAL#0.00326013840564205, LREAL#-0.0031732974749522345, LREAL#0.003127980724725045, LREAL#-0.0029403086218353475, LREAL#0.003000464472349495, LREAL#-0.0027155024267765749, LREAL#0.0028774266397613383, LREAL#-0.00249859151168035, LREAL#0.0027587099431366047, LREAL#-0.0022892985912802669, LREAL#0.0026441626225196632, LREAL#-0.0020873561186750315, LREAL#0.0025336382478228429, LREAL#-0.0018925059433133396, LREAL#0.0024269955316394355, LREAL#-0.0017044989809904649, LREAL#0.0023240981486307415, LREAL#-0.001523094895434662, LREAL#0.002224814561256352, LREAL#-0.0013480617910764175, LREAL#0.0021290178516248127, LREAL#-0.0011791759166077203, LREAL#0.0020365855592498149, LREAL#-0.0010162213789525075, LREAL#0.0019473995245043718, LREAL#-0.00085898986728249538, LREAL#0.001861345737573008, LREAL#-0.0007072803867257466, LREAL#0.0017783141927087897, LREAL#-0.00056089900142747685, LREAL#0.0016981987476088775, LREAL#-0.00041965858663463735, LREAL#0.0016208969877289099, LREAL#-0.00028337858948742907, LREAL#0.0015463100953626583, LREAL#-0.00015188479821185292, LREAL#0.0014743427233197589, LREAL#-2.5009119418409047E-5, LREAL#0.0014049028730397563, LREAL#9.7410636778025238E-5, LREAL#0.0013379017769870371, LREAL#0.00021553096409143352, LREAL#0.0012732537851759288, LREAL#0.000329502860116448, LREAL#0.0012108762556811894, LREAL#0.00043947201935413038, LREAL#0.0011506894489937236, LREAL#0.00054557901945870171, LREAL#0.0010926164260866547, LREAL#0.00064795950094312838, LREAL#0.0010365829500613034, LREAL#0.00074674434057342887, LREAL#0.00098251739124740776, LREAL#0.00084205981867329651, LREAL#0.00093035063563620636, LREAL#0.00093402778055297483, LREAL#0.00088001599652954383, LREAL#0.0010227657922685272, LREAL#0.00083144912929171259, LREAL#0.0011083872909109674, LREAL#0.00078458794909530951, LREAL#0.0011910017296171095, LREAL#0.00073937255155595658, LREAL#0.0012707147174875113, LREAL#0.00069574513615428349, LREAL#0.0013476281545905262, LREAL#0.00065364993234734426, LREAL#0.0014218403622249763, LREAL#0.00061303312827511679, LREAL#0.0014934462086078622, LREAL#0.000573842801970774, LREAL#0.0015625372301479527, LREAL#0.00053602885498692612, LREAL#0.0016292017484601563, LREAL#0.00049954294835288934, LREAL#0.0016935249832703426, LREAL#0.00046433844078121357, LREAL#0.0017555891613548523, LREAL#0.00043037032904441152, LREAL#0.0018154736216540179, LREAL#0.000397595190445604, LREAL#0.001873254916694134, LREAL#0.00036597112730973489, LREAL#0.0019290069104473311, LREAL#0.00033545771342420448, LREAL#0.0019828008727546453, LREAL#0.00030601594236050439, LREAL#0.0020347055704329387, LREAL#0.00027760817761090639, LREAL#0.0020847873551820164, LREAL#0.00025019810447631717, LREAL#0.0021331102484044677, LREAL#0.00022375068364378456, LREAL#0.0021797360230466673, LREAL#0.0001982321063944995, LREAL#0.0022247242825653669, LREAL#0.00017360975138492105, LREAL#0.0022681325371209393];
  END_VAR

            

CASE ssMethodType OF
    SINT#0: 
        (* SystemInitialize for Atomic SubSystem: '<Root>/MPC DMC' *)
        (* InitializeConditions for UnitDelay: '<S1>/Unit Delay' *)
        UnitDelay_DSTATE := LREAL#0.0;
        (* InitializeConditions for DiscreteTransferFcn: '<S1>/Discrete Transfer Fcn1' *)
        DiscreteTransferFcn1_states := LREAL#0.0;
        (* End of SystemInitialize for SubSystem: '<Root>/MPC DMC' *)
        (* '<S2>:1:12' d_hist    = zeros(Ntop, 1); *)
        (* SystemInitialize for Atomic SubSystem: '<Root>/MPC DMC' *)
        (* SystemInitialize for MATLAB Function: '<S1>/Calculating Free Response' *)

        FOR i := DINT#0 TO DINT#147 DO 
            d_hist[i] := LREAL#0.0;
        END_FOR;

        (* End of SystemInitialize for SubSystem: '<Root>/MPC DMC' *)
        (* oldest..newest, IC = 0 *)
        (* '<S2>:1:13' u100_hist = zeros(bigDelay, 1); *)
        (* SystemInitialize for Atomic SubSystem: '<Root>/MPC DMC' *)
        (* SystemInitialize for MATLAB Function: '<S1>/Calculating Free Response' *)

        FOR i := DINT#0 TO DINT#99 DO 
            u100_hist[i] := LREAL#0.0;
        END_FOR;

        (* End of SystemInitialize for SubSystem: '<Root>/MPC DMC' *)
        (* z^-100 delay line, IC = 0 *)
        (* '<S2>:1:14' w_hist    = zeros(Nbot - 1, 1); *)
        (* SystemInitialize for Atomic SubSystem: '<Root>/MPC DMC' *)
        (* SystemInitialize for MATLAB Function: '<S1>/Calculating Free Response' *)

        FOR i := DINT#0 TO DINT#48 DO 
            w_hist[i] := LREAL#0.0;
        END_FOR;

        (* 49-sample history for Tapped Delay1 *)
        (* '<S2>:1:15' u_prev    = 0; *)
        u_prev_f := LREAL#0.0;
        (* End of SystemInitialize for SubSystem: '<Root>/MPC DMC' *)
        (* previous u, for Difference1 *)
        (* '<S3>:1:12' u150_hist = zeros(N, 1); *)
        (* SystemInitialize for Atomic SubSystem: '<Root>/MPC DMC' *)
        (* SystemInitialize for MATLAB Function: '<S1>/Model' *)

        FOR i := DINT#0 TO DINT#149 DO 
            u150_hist[i] := LREAL#0.0;
        END_FOR;

        (* End of SystemInitialize for SubSystem: '<Root>/MPC DMC' *)
        (* z^-150 delay line, IC = 0 *)
        (* '<S3>:1:13' du_hist   = zeros(N - 1, 1); *)
        (* SystemInitialize for Atomic SubSystem: '<Root>/MPC DMC' *)
        (* SystemInitialize for MATLAB Function: '<S1>/Model' *)

        FOR i := DINT#0 TO DINT#148 DO 
            du_hist[i] := LREAL#0.0;
        END_FOR;

        (* 149-sample history (oldest..newest), IC = 0 *)
        (* '<S3>:1:14' u_prev    = 0; *)
        u_prev := LREAL#0.0;
        (* End of SystemInitialize for SubSystem: '<Root>/MPC DMC' *)
        (* previous u, for Difference *)
    SINT#1: 
        (* Outputs for Atomic SubSystem: '<Root>/MPC DMC' *)
        (* MATLAB Function: '<S1>/Calculating Free Response' incorporates:
         *  UnitDelay: '<S1>/Unit Delay' *)
        (* MATLAB Function 'MPC DMC/Calculating Free Response': '<S2>:1' *)
        (* '<S2>:1:2' Ntop = 148; *)
        (* '<S2>:1:3' Nbot = 50; *)
        (* '<S2>:1:4' bigDelay = 100; *)
        (* ---- lazy init on first call only ---- *)
        (* Codegen only allows reading a persistent variable via isempty(...) *)
        (* before it has been assigned; we never read its value before this. *)
        (* '<S2>:1:11' if isempty(d_hist) *)
        (* ---- top branch ---- *)
        (* '<S2>:1:19' d_k = u_k - u_prev; *)
        d_k := UnitDelay_DSTATE - u_prev_f;
        (* Difference1: (z-1)/z *)
        (* '<S2>:1:20' u_prev = u_k; *)
        u_prev_f := UnitDelay_DSTATE;
        (* End of Outputs for SubSystem: '<Root>/MPC DMC' *)
        (* update for next call *)
        (* '<S2>:1:22' v_raw = d_hist; *)
        (* oldest->newest, 148x1 (most recent 148 past d's) *)
        (* '<S2>:1:23' v = flipud(v_raw); *)
        (* Outputs for Atomic SubSystem: '<Root>/MPC DMC' *)
        (* MATLAB Function: '<S1>/Calculating Free Response' incorporates:
         *  UnitDelay: '<S1>/Unit Delay' *)

        FOR i := DINT#0 TO DINT#147 DO 
            v[i] := d_hist[i];
        END_FOR;


        FOR i := DINT#0 TO DINT#73 DO 
            xtmp := v[i];
            v[i] := v[DINT#147 - i];
            v[DINT#147 - i] := xtmp;
        END_FOR;

        (* Selector reverse -> newest->oldest *)
        (* '<S2>:1:24' y1 = H * v; *)
        (* 50x1 *)
        (* '<S2>:1:26' d_hist = [d_hist(2:end); d_k]; *)

        FOR i := DINT#0 TO DINT#146 DO 
            d_hist[i] := d_hist[i + DINT#1];
        END_FOR;

        d_hist[DINT#147] := d_k;
        (* shift in new sample, drop oldest *)
        (* ---- bottom branch ---- *)
        (* '<S2>:1:29' u100_k = u100_hist(1); *)
        u100_k := u100_hist[DINT#0];
        (* oldest entry = u[k-100] *)
        (* '<S2>:1:30' u100_hist = [u100_hist(2:end); u_k]; *)

        FOR i := DINT#0 TO DINT#98 DO 
            u100_hist[i] := u100_hist[i + DINT#1];
        END_FOR;

        u100_hist[DINT#99] := UnitDelay_DSTATE;
        (* shift in current u, drop oldest *)
        (* '<S2>:1:32' w = [w_hist; u100_k]; *)

        FOR i := DINT#0 TO DINT#48 DO 
            w[i] := w_hist[i];
        END_FOR;

        w[DINT#49] := u100_k;
        (* oldest..newest, current (u100_k) last, 50x1 *)
        (* '<S2>:1:33' y2 = SS_N1 .* w; *)
        (* 50x1 *)
        (* '<S2>:1:35' w_hist = [w_hist(2:end); u100_k]; *)

        FOR i := DINT#0 TO DINT#47 DO 
            w_hist[i] := w_hist[i + DINT#1];
        END_FOR;

        w_hist[DINT#48] := u100_k;
        (* MATLAB Function: '<S1>/Model' incorporates:
         *  UnitDelay: '<S1>/Unit Delay' *)
        (* shift in u100_k, drop oldest, for next call *)
        (* ---- combine ---- *)
        (* '<S2>:1:38' f = y1 + y2; *)
        (* 50x1 *)
        (* MATLAB Function 'MPC DMC/Model': '<S3>:1' *)
        (* '<S3>:1:3' N = 150; *)
        (* number of taps / delay length, matches z^-150 and 149+1 taps *)
        (* '<S3>:1:7' SS_1N  = SS(1:N); *)
        (* 1x150 row vector — feeds the "SS(1:N)*u" gain *)
        (* '<S3>:1:8' SS_N1  = SS(N+1); *)
        (* scalar — feeds both "SS(N+1)" gains (ss_gain in the other block too) *)
        (* ---- lazy init on first call only (isempty check is codegen-legal) ---- *)
        (* '<S3>:1:11' if isempty(u150_hist) *)
        (* '<S3>:1:17' if numel(SS_1N) ~= N *)
        (* '<S3>:1:21' if ~isscalar(SS_N1) *)
        (* '<S3>:1:25' SS_1N_row = reshape(SS_1N, 1, N); *)
        (* ensure 1xN row for the dot product *)
        (* ---- top branch ---- *)
        (* '<S3>:1:28' u150_k = u150_hist(1); *)
        u150_k := u150_hist[DINT#0];
        (* oldest entry = u[k-N] *)
        (* '<S3>:1:29' y1 = SS_N1 * u150_k; *)
        (* scalar *)
        (* '<S3>:1:31' u150_hist = [u150_hist(2:end); u_k]; *)
        (* shift in current u, drop oldest *)
        (* ---- bottom branch ---- *)
        (* '<S3>:1:34' du_k = u_k - u_prev; *)
        du_k := UnitDelay_DSTATE - u_prev;
        (* Difference: (z-1)/z *)
        (* '<S3>:1:35' u_prev = u_k; *)
        u_prev := UnitDelay_DSTATE;
        (* End of Outputs for SubSystem: '<Root>/MPC DMC' *)
        (* w = [du_k, du(k-1), ..., du(k-149)], newest->oldest, current first *)
        (* '<S3>:1:38' w = [du_k; flipud(du_hist)]; *)
        (* Outputs for Atomic SubSystem: '<Root>/MPC DMC' *)
        (* MATLAB Function: '<S1>/Model' incorporates:
         *  UnitDelay: '<S1>/Unit Delay' *)

        FOR i := DINT#0 TO DINT#148 DO 
            u150_hist[i] := u150_hist[i + DINT#1];
            x[i] := du_hist[i];
        END_FOR;

        u150_hist[DINT#149] := UnitDelay_DSTATE;

        FOR i := DINT#0 TO DINT#73 DO 
            xtmp := x[i];
            x[i] := x[DINT#148 - i];
            x[DINT#148 - i] := xtmp;
        END_FOR;

        (* 150x1 *)
        (* '<S3>:1:40' y2 = SS_1N_row * w; *)
        (* 1x150 * 150x1 -> scalar *)
        (* '<S3>:1:42' du_hist = [du_hist(2:end); du_k]; *)

        FOR i := DINT#0 TO DINT#147 DO 
            du_hist[i] := du_hist[i + DINT#1];
        END_FOR;

        du_hist[DINT#148] := du_k;
        (* End of Outputs for SubSystem: '<Root>/MPC DMC' *)
        (* shift in current du, drop oldest *)
        (* ---- combine ---- *)
        (* '<S3>:1:45' ym = y1 + y2; *)
        (* scalar *)
        (* Outputs for Atomic SubSystem: '<Root>/MPC DMC' *)
        (* MATLAB Function: '<S1>/Model' *)
        du_k_0[DINT#0] := du_k;

        FOR i := DINT#0 TO DINT#148 DO 
            du_k_0[i + DINT#1] := x[i];
        END_FOR;

        rtb_u := LREAL#0.0;

        FOR i := DINT#0 TO DINT#149 DO 
            rtb_u := (Model_SS[i] * du_k_0[i]) + rtb_u;
        END_FOR;

        (* Sum: '<S1>/Sum2' incorporates:
         *  MATLAB Function: '<S1>/Model' *)
        xtmp := y - ((LREAL#19.906243860199364 * u150_k) + rtb_u);
        (* Gain: '<S1>/Gain1' *)
        rtb_Gain1_idx_0 := LREAL#0.0;

        FOR i := DINT#0 TO DINT#49 DO 
            (* MATLAB Function: '<S1>/Calculating Free Response' *)
            rtb_u := LREAL#0.0;

            FOR i_0 := DINT#0 TO DINT#147 DO 
                rtb_u := (CalculatingFreeResponse_H[(DINT#50 * i_0) + i] * v[i_0]) + rtb_u;
            END_FOR;

            (* Gain: '<S1>/Gain1' incorporates:
             *  MATLAB Function: '<S1>/Calculating Free Response'
             *  Sum: '<S1>/Sum'
             *  Sum: '<S1>/Sum3' *)
            rtb_Gain1_idx_0 := (Gain1_Gain[i * DINT#2] * (b_r - (((LREAL#19.906243860199364 * w[i]) + rtb_u) + xtmp))) + rtb_Gain1_idx_0;
        END_FOR;

        (* Saturate: '<S1>/Saturation' incorporates:
         *  Fcn: '<S1>/Fcn'
         *  Gain: '<S1>/Gain1' *)

        IF rtb_Gain1_idx_0 > LREAL#0.2 THEN 
            xtmp := LREAL#0.2;
        ELSIF rtb_Gain1_idx_0 >= LREAL#-0.2 THEN 
            xtmp := rtb_Gain1_idx_0;
        ELSE 
            xtmp := LREAL#-0.2;
        END_IF;

        (* End of Saturate: '<S1>/Saturation' *)
        

        (* DiscreteTransferFcn: '<S1>/Discrete Transfer Fcn1' *)
        rtb_u := xtmp - ( -DiscreteTransferFcn1_states);
        (* Saturate: '<S1>/Saturation1' incorporates:
         *  DiscreteTransferFcn: '<S1>/Discrete Transfer Fcn1' *)

        IF rtb_u > LREAL#0.9 THEN 
            xtmp := LREAL#0.9;
        ELSIF rtb_u >= LREAL#0.1 THEN 
            xtmp := rtb_u;
        ELSE 
            xtmp := LREAL#0.1;
        END_IF;

        (* End of Saturate: '<S1>/Saturation1' *)
        

        (* Update for UnitDelay: '<S1>/Unit Delay' incorporates:
         *  DiscreteTransferFcn: '<S1>/Discrete Transfer Fcn1' *)
        UnitDelay_DSTATE := rtb_u;
        (* Update for DiscreteTransferFcn: '<S1>/Discrete Transfer Fcn1' *)
        DiscreteTransferFcn1_states := rtb_u;
        (* Outport: '<Root>/u' incorporates:
         *  Gain: '<S1>/Gain' *)
        u := LREAL#100.0 * xtmp;
        (* End of Outputs for SubSystem: '<Root>/MPC DMC' *)
END_CASE;



          
END_FUNCTION_BLOCK
